			(* Case 157 - Attesa distacco lastra *)					
			157:
				IF Programma_Z[Z_PosDistaccoLastraInLentaLastra].Stato = INTERROTTO	THEN
					Ciclo^.Passo := 157;																
				ELSE
					TFTimerSet(ADR(TimerAttesaCadutaLastra),HMI_TempoAttesaPartenzaDopoPrelievo, Programma_Z[Z_PosDistaccoLastraInLentaLastra].Stato <> TERMINATO);		
					IF Programma_Z[Z_PosDistaccoLastraInLentaLastra].Stato = TERMINATO AND TFTimerDone(ADR(TimerAttesaCadutaLastra)) THEN
						TFParametersArrayClear(ADR(ParametersArray));
						TFCommandSend(CmdCheckPresence,ParametersArray,Modules^.Pinza.Cmd);
						Ciclo^.Passo := 158;	
					END_IF
				END_IF	
					
			(* Case 158 -  Attesa completamento del comando *)
			158: 
				IF Programma_Z[Z_PosDistaccoLastraInLentaLastra].Stato = INTERROTTO	THEN
					Ciclo^.Passo := 158;																
				ELSE
					//TFTimerSet(ADR(TimerAttesaCadutaLastra),HMI_TempoAttesaPartenzaDopoPrelievo, (Programma_Z[Z_PosDistaccoLastraInLentaLastra].Stato <> TERMINATO));
					IF Programma_Z[Z_PosDistaccoLastraInLentaLastra].Stato = TERMINATO AND 
						TFTimerDone(ADR(TimerAttesaCadutaLastra)) AND
						TFStateCodeGet(Modules^.Pinza.State) = StateCHECKPRESENCE_END THEN
						IF Modules^.Pinza.StatoPinza.ElementoPrelevato THEN
							Ciclo^.Passo := 1000;	//CICLO TERMINATO
							Modules^.Ax_J.IN_Stop := TRUE; //Fermo Comando di tasteggio
							STEPDone := FALSE;
						ELSIF NOT Modules^.Pinza.StatoPinza.ElementoPrelevato THEN
							//IF NumeroTentativiPresaAttuali >= NumeroTentativiPresa THEN
								Errore := ErrMalfunzionamentoSensoriPresenzaPinza;
								//IF StepInto THEN
								//	Ciclo^.Passo 		:= 1000;//CICLO TERMINATO
								//	STEPDone 			:= FALSE;
								//END_IF
							//ELSE
								//Ciclo^.Passo := 150;//torno a fare prelievo
							//	NumeroTentativiPresaAttuali := NumeroTentativiPresaAttuali+1;
							//END_IF
						END_IF	
					END_IF
				END_IF	

			(* Case 1000 *)
			1000:
				STEPDone := TRUE;
				Ciclo^.Stato := TERMINATO;
				Ciclo^.Passo := 1000;
				
			(* Case 9999 - Ciclo NON annullato o NON terminato*)
			9999:
				Ciclo^.Stato := INTERROTTO;
				Ciclo^.Passo := 9999;
	ELSE						
		;	
	END_CASE;
ELSE								//Se il ciclo deve essere interrotto, setto il suo nuovo stato
	Ciclo^.Stato := INTERROTTO;
END_IF
END_ACTION

ACTION Verticale:
TFTimerCall(ADR(TimerAttesaCadutaLastra),TimeBase);
TFTimerCall(ADR(ReControlPiezaCogida),TimeBase); 
TFTimerCall(ADR(ReMovEjeX),TimeBase); 
(* Set della variabile che mi permette di fare lo STEP nel ciclo *)
StepInto := (Abilita_Ciclo_Step AND Command_Step) OR NOT Abilita_Ciclo_Step;

(* Reset Anticipo Dinamico se non ho l'abilitazione *)
IF NOT AbilitazioneAnticipoDinamicoMovimenti OR NOT HMI_DisabilitaAnticipiGLOBALE THEN
	QuotaAnticipoDinamicaX_Raggiunta := FALSE;
	QuotaAnticipoDinamicaY_Raggiunta := FALSE;
	QuotaAnticipoDinamicaZ_Raggiunta := FALSE;
END_IF
//
//
AttivazioneVuotoDistanza := TRUE;

IF Ciclo^.Passo = 116 THEN
Temp_INT[9] := 	Temp_INT[9] + 1;
TFTimerSet(ADR(ReControlPiezaCogida),10000, FALSE );	
ELSE
TFTimerSet(ADR(ReControlPiezaCogida),10000, TRUE );	
END_IF

IF Ciclo^.Passo = 27 THEN

TFTimerSet(ADR(ReMovEjeX),1000, FALSE );	
ELSE
TFTimerSet(ADR(ReMovEjeX),1000, 
TFAsseInFinestra(Posizione_Attuale := Modules^.AX_Y.Ax^.AxRef^.NcToPlc.ActPos ,
 Posizione_Finale := Programma_Y[Y_PosFuoriIngombroVuotoLastra].Quota_Destinazione ,FinestraDiControllo := 30.0 ) );	
END_IF

EjeYPosFueraIngombro := TFAsseInFinestra(Posizione_Attuale := Modules^.AX_Y.Ax^.AxRef^.NcToPlc.ActPos ,
 Posizione_Finale := Programma_Y[Y_PosFuoriIngombroVuotoLastra].Quota_Destinazione ,FinestraDiControllo := 30.0 );

EjeYPos0Ingombro :=  TFAsseInFinestra(Posizione_Attuale := Modules^.AX_Y.Ax^.AxRef^.NcToPlc.ActPos ,
 Posizione_Finale := Programma_Y[Y_PosPasillo0grados].Quota_Destinazione ,FinestraDiControllo := 30.0 ) ;
 
EjeYPos180Ingombro := TFAsseInFinestra(Posizione_Attuale := Modules^.AX_Y.Ax^.AxRef^.NcToPlc.ActPos ,
 Posizione_Finale := Programma_Y[Y_PosPasillo180grados].Quota_Destinazione ,FinestraDiControllo := 30.0 ) ;





Temp_Bool[58]:= TFAsseInFinestra(Posizione_Attuale := Modules^.AX_Y.Ax^.AxRef^.NcToPlc.ActPos ,
 Posizione_Finale := Programma_Y[Y_PosFuoriIngombroVuotoLastra].Quota_Destinazione ,FinestraDiControllo := 30.0 ) OR

(( TFAsseInFinestra(Posizione_Attuale := Modules^.AX_Y.Ax^.AxRef^.NcToPlc.ActPos ,
 Posizione_Finale := Programma_Y[Y_PosPasillo0grados].Quota_Destinazione ,FinestraDiControllo := 30.0 ) OR

TFAsseInFinestra(Posizione_Attuale := Modules^.AX_Y.Ax^.AxRef^.NcToPlc.ActPos ,
 Posizione_Finale := Programma_Y[Y_PosPasillo180grados].Quota_Destinazione ,FinestraDiControllo := 30.0 )) (*AND RobotWorkAreaCavallete (*AND MultiplesCavalletesReceta *) *))  ;

 
 
 
Temp_Bool[25] := TFTimerDone(ADR(ReControlPiezaCogida));

//Valuto l'angolo di J per stabilire se è "inclinata"

PinzaVerticale 	:= Modules^.AX_J.Ax^.Status.ActPosition > 95 OR Modules^.AX_J.Ax^.Status.ActPosition < 85;
PinzaInPresa	:= Modules^.Pinza.StatoPinza.LatoDxPiastrellaInPresa AND Modules^.Pinza.StatoPinza.LatoSxPiastrellaInPresa;


IF NOT InterrompiCiclo THEN
	IF Ciclo^.Stato = TERMINATO OR Ciclo^.Stato = ANNULLATO THEN
		Ciclo^.Passo 	:= 0;
		Errore 			:= 0;
	ELSIF Ciclo^.Stato = INTERROTTO THEN
		Ciclo^.Passo 	:= 9999;
	END_IF
	CASE Ciclo^.Passo OF

			(* Case 0 *)
			0:  Ciclo^.Stato 		:= IN_ESECUZIONE;
				ReqStartAspirazione := FALSE;
				STEPDone 			:= FALSE;
				PosicionJSalida    := 0 ;
				
				IF Modules^.Pinza.CmdNext.Code = '' AND NOT PinzaInPresa THEN
					TFParametersArrayClear(ADR(ParametersArray));
					IF InWaitPosition THEN
						Modules^.Pinza.IN.RichiestaRicalibrazioneOvemEsterna := TRUE; //Ricalibrazione automatica OVEM
					END_IF
					TFCommandSend(CmdUNLOAD,ParametersArray,Modules^.Pinza.Cmd);
					Ciclo^.Passo := 11;
				ELSIF PinzaInPresa THEN
					Errore := ErrPRESENZA_MATERIALE_SUPINZA_CICLO_PRELPACCO;
				END_IF
				(* Start tempo ciclo *)
				
			(* Case 11 - Attesa comando temrinato pinza *)
			11:			
				IF TFStateCodeGet(Modules^.Pinza.State) = StateUNLOAD_END THEN
					Ciclo^.Passo := 12;	
				ELSIF TFStateCodeGet(Modules^.Pinza.State) = StateError THEN
					Ciclo^.Passo := 11;																
				END_IF
				
			(* Case 12 - Blocca Rotazione e Basculante *)
			12:
				IF TFStateCodeGet(Modules^.Pinza.State) = StateError THEN
					Ciclo^.Passo := 12;																
				ELSE
					//TFParametersArrayClear(ADR(ParametersArray));
					//TFCommandSend(CmdBloccaPinza,ParametersArray,Modules^.Pinza.Cmd);
					Ciclo^.Passo := 13;
				END_IF				

			(* Case 13 - Blocca Rotazione e Basculante *)
			13:
				IF TFStateCodeGet(Modules^.Pinza.State) = StateError THEN
					Ciclo^.Passo := 13;																
				ELSE
					//IF TFStateCodeGet(Modules^.Pinza.State) = StateBloccaPinza_END THEN//Pinza bloccata
						Ciclo^.Passo := 20;
					//END_IF	
				END_IF	
	
			(* Case 20 - TRASLAZIONE A QUOTA DI FUORI INGOMBRO *)	
			20:	
				//IF TFStateCodeGet(Modules^.Pinza.State) = StateUNLOAD_END THEN
					IF StepInto THEN
						Programma_Z[Z_PosFuoriIngombroVuotoLastra].Stato 			:= DA_ESEGUIRE;
						Programma_Z[Z_PosFuoriIngombroVuotoLastra].InterpolaAsse 	:= NO_INTERPOLAZIONE_ASSE;
						ProgrammaToModule_Z 										:= Programma_Z[Z_PosFuoriIngombroVuotoLastra];
						Ciclo^.Passo := 21;
						STEPDone := FALSE;
						
					(*	Programma_Z[Z_PosFuoriIngombroCaricoLastra].Stato 			:= DA_ESEGUIRE;
						Programma_Z[Z_PosFuoriIngombroCaricoLastra].InterpolaAsse 	:= NO_INTERPOLAZIONE_ASSE;
						ProgrammaToModule_Z 										:= Programma_Z[Z_PosFuoriIngombroCaricoLastra];
						Ciclo^.Passo := 21;
						STEPDone := FALSE; *)
					END_IF
				//END_IF
				
			(* Case 21 - Attesa completamento del comando MOVETOPOS o del raggiungimento quota di Pre-Movimento se abilitata la funzione*)
			21: 
					
				//IF Programma_Z[Z_PosFuoriIngombroCaricoLastra].Stato = INTERROTTO THEN
				IF Programma_Z[Z_PosFuoriIngombroVuotoLastra].Stato = INTERROTTO THEN
					Ciclo^.Passo := 21;		
				//ELSIF Programma_Z[Z_PosFuoriIngombroCaricoLastra].Stato = TERMINATO OR
				ELSIF Programma_Z[Z_PosFuoriIngombroVuotoLastra].Stato = TERMINATO OR
					Asse_Z_InFinestraDiPassMode THEN
					IF PinzaVerticale THEN//Se la pinza è già verticale in finestra di prelievo

						IF Modules^.AX_Y.Ax^.AxRef^.NcToPlc.ActPos <= Programma_Y[Y_PosFuoriIngombroVuotoLastra].Quota_Destinazione AND NOT RobotWorkAreaCavallete THEN
							Programma_Y[Y_PosFuoriIngombroVuotoLastra].Stato 				:= DA_ESEGUIRE;
							//Programma_Y[Y_PosFuoriIngombroVuotoLastra].InterpolaAsse 		:= INTERPOLAZIONE_ASSE;
							Programma_Y[Y_PosFuoriIngombroVuotoLastra].InterpolaAsse 		:= No_INTERPOLAZIONE_ASSE;
							ProgrammaToModule_Y 									:= Programma_Y[Y_PosFuoriIngombroVuotoLastra];
							
							Programma_J[J_PosFuoriIngombroPosAttuale].Stato 		:= DA_ESEGUIRE;
							//Programma_J[J_PosFuoriIngombroPosAttuale].InterpolaAsse := INTERPOLAZIONE_ASSE;
							Programma_J[J_PosFuoriIngombroPosAttuale].InterpolaAsse := No_INTERPOLAZIONE_ASSE;
							ProgrammaToModule_J 									:= Programma_J[J_PosFuoriIngombroPosAttuale];
	
							StartInterpolazioneAssi^ 								:= TRUE;
							Ciclo^.Passo := 22; 
							STEPDone := TRUE;	
						ELSE
							Ciclo^.Passo := 23; 
							STEPDone := TRUE;	
						END_IF						
					ELSIF NOT PinzaVerticale THEN
						Ciclo^.Passo := 25; 
						STEPDone := TRUE;							
					ELSE
						Ciclo^.Passo := 21;		
						Errore := 1;
					END_IF
				END_IF
			
			(* Case 21 - Rotazione Asse K *)	
			22: IF Programma_Z[Z_PosFuoriIngombroVuotoLastra].Stato = INTERROTTO OR
					Programma_Y[Y_PosFuoriIngombroVuotoLastra].Stato = INTERROTTO OR
					Programma_J[J_PosFuoriIngombroPosAttuale].Stato = INTERROTTO THEN
					 Ciclo^.Passo := 22;
				ELSIF Programma_Z[Z_PosFuoriIngombroVuotoLastra].Stato = TERMINATO AND //OR Asse_Z_InFinestraDiPassMode) AND 
					Programma_Y[Y_PosFuoriIngombroVuotoLastra].Stato = TERMINATO AND//OR Asse_Y_InFinestraDiPassMode) AND
					Programma_J[J_PosFuoriIngombroPosAttuale].Stato = TERMINATO THEN//OR Asse_J_InFinestraDiPassMode) THEN
						IF StepInto THEN
							Ciclo^.Passo := 23;
							STEPDone := FALSE;
						END_IF									
				END_IF

			(* Case 23 - Attesa completamento comandi *)	
			23: 	
				STEPDone := TRUE;
				Ciclo^.Passo := 24;
	
			(* Case 24 - free *)	
			24:	
				STEPDone := FALSE;
				Ciclo^.Passo := 25;
			
			(* Case 25 - Vado a quota di CORRIDOIO PER ROTAZIONE con Y *)
			25:	IF Programma_Z[Z_PosFuoriIngombroVuotoLastra].Stato = INTERROTTO THEN
					Ciclo^.Passo := 25;										
				ELSE
					
					IF StepInto THEN
							//IF 	Programma_Z[Y_PosFuoriIngombroVuotoLastra].Stato = TERMINATO THEN
							IF 	Programma_Z[Z_PosFuoriIngombroVuotoLastra].Stato = TERMINATO  THEN
								PruLineaContactos := (PosRobot = NuPosGuiroPiking  AND PikingConCavallete) 
												OR (( NOT MultiplesCavalletesReceta 
												OR PosicionJDestino = PosicionJOrigen) AND NOT PikingConCavallete) ;
							
								
										
								(*
									Programma_X[X_PosStartLentaPrelievoLastra].Stato 			:= DA_ESEGUIRE;
									//Programma_X[X_PosStartLentaPrelievoLastra].InterpolaAsse 	:= INTERPOLAZIONE_ASSE;
									Programma_X[X_PosStartLentaPrelievoLastra].InterpolaAsse 	:= No_INTERPOLAZIONE_ASSE;
									ProgrammaToModule_X 										:= Programma_X[X_PosStartLentaPrelievoLastra];
								*)
								
								
								IF (AngulosDiferentes OR PosicionJDestino <> PosicionJActual)  AND (RobotWorkAreaCavallete OR MultiplesCavalletesReceta) THEN 
									Temp_UINT [1] := Temp_UINT [1]+1;
									IF PosicionJActual = 0 THEN
										(*
										//********************************************************************
										Programma_Y[Y_PosFuoriIngombroVuotoLastra].Stato 	:= NON_ESEGUITO;
										Programma_Y[Y_PosPasillo180grados].Stato 			:= NON_ESEGUITO;
										Programma_Y[Y_PosgiroPieza].Stato 					:= NON_ESEGUITO ;
										//*********************************************************************
										*)
										Programma_Y[Y_PosPasillo0grados].Stato 			:= DA_ESEGUIRE;
										Programma_Y[Y_PosPasillo0grados].InterpolaAsse 	:= INTERPOLAZIONE_ASSE;
										ProgrammaToModule_Y 							:= Programma_Y[Y_PosPasillo0grados];
										
										Programma_J[Pos0TrasporteCavallete].Stato 						:= DA_ESEGUIRE;
										Programma_J[Pos0TrasporteCavallete].InterpolaAsse 				:= No_INTERPOLAZIONE_ASSE;
										ProgrammaToModule_J 											:= Programma_J[Pos0TrasporteCavallete];	
										IF Temp_Bool[50] THEN
											StartInterpolazioneAssi^ := TRUE;
											Ciclo^.Passo := 27;
										END_IF
										
									END_IF
									IF PosicionJActual = 180 THEN
										Programma_Y[Y_PosPasillo180grados].Stato 			:= DA_ESEGUIRE;
										Programma_Y[Y_PosPasillo180grados].InterpolaAsse 	:= INTERPOLAZIONE_ASSE;
										ProgrammaToModule_Y 								:= Programma_Y[Y_PosPasillo180grados];
										
										Programma_J[Pos180TrasporteCavallete].Stato 						:= DA_ESEGUIRE;
										Programma_J[Pos180TrasporteCavallete].InterpolaAsse 				:= No_INTERPOLAZIONE_ASSE;
										ProgrammaToModule_J 											:= Programma_J[Pos180TrasporteCavallete];
										IF Temp_Bool[50] THEN
											StartInterpolazioneAssi^ := TRUE;
											Ciclo^.Passo := 27;
										END_IF
									END_IF
									
									IF PosicionJActual = 90 AND PosicionJOrigen = 0 THEN
										Programma_Y[Y_PosPasillo0grados].Stato 			:= DA_ESEGUIRE;
										Programma_Y[Y_PosPasillo0grados].InterpolaAsse 	:= INTERPOLAZIONE_ASSE;
										ProgrammaToModule_Y 								:= Programma_Y[Y_PosPasillo0grados];
										
										Programma_J[Pos0TrasporteCavallete].Stato 						:= DA_ESEGUIRE;
										Programma_J[Pos0TrasporteCavallete].InterpolaAsse 				:= No_INTERPOLAZIONE_ASSE;
										ProgrammaToModule_J 											:= Programma_J[Pos0TrasporteCavallete];
										IF Temp_Bool[50] THEN
											StartInterpolazioneAssi^ := TRUE;
											Ciclo^.Passo := 27;
										END_IF
									END_IF
									IF PosicionJActual = 90 AND PosicionJOrigen = 180 THEN
										Programma_Y[Y_PosPasillo180grados].Stato 			:= DA_ESEGUIRE;
										Programma_Y[Y_PosPasillo180grados].InterpolaAsse 	:= INTERPOLAZIONE_ASSE;
										ProgrammaToModule_Y 								:= Programma_Y[Y_PosPasillo180grados];
										
										Programma_J[Pos180TrasporteCavallete].Stato 						:= DA_ESEGUIRE;
										Programma_J[Pos180TrasporteCavallete].InterpolaAsse 				:= No_INTERPOLAZIONE_ASSE;
										ProgrammaToModule_J 											:= Programma_J[Pos180TrasporteCavallete];
										IF Temp_Bool[50] THEN
											StartInterpolazioneAssi^ := TRUE;
											Ciclo^.Passo := 27;
										END_IF
									END_IF
									//PosicionJSalida := PosicionJActual ;
								ELSIF NOT AngulosDiferentes AND RobotWorkAreaCavallete AND PosicionJDestino = PosicionJActual  THEN
										Temp_UINT [2] := Temp_UINT [2]+1;
										Programma_Y[Y_PosFuoriIngombroVuotoLastra].Stato 				:= DA_ESEGUIRE;
										Programma_Y[Y_PosFuoriIngombroVuotoLastra].InterpolaAsse 		:= No_INTERPOLAZIONE_ASSE;
										//Programma_Y[Y_PosFuoriIngombroVuotoLastra].InterpolaAsse 		:= INTERPOLAZIONE_ASSE;
										ProgrammaToModule_Y 										:= Programma_Y[Y_PosFuoriIngombroVuotoLastra];
										
										Programma_J[J_PosFuoriIngombro].Stato 						:= DA_ESEGUIRE;
										//Programma_J[J_PosFuoriIngombro].InterpolaAsse 				:= INTERPOLAZIONE_ASSE;
										Programma_J[J_PosFuoriIngombro].InterpolaAsse 				:= No_INTERPOLAZIONE_ASSE;
										ProgrammaToModule_J 										:= Programma_J[J_PosFuoriIngombro];
										IF Temp_Bool[50] THEN
											StartInterpolazioneAssi^ := TRUE;
											Ciclo^.Passo := 27;
										END_IF
										
								ELSIF  (PosRobot = NuPosGuiroPiking  AND PikingConCavallete) OR (( NOT MultiplesCavalletesReceta OR PosicionJDestino = PosicionJOrigen) AND NOT PikingConCavallete)   THEN
										Temp_UINT [3] := Temp_UINT [3]+1;
								
										Programma_Y[Y_PosFuoriIngombroVuotoLastra].Stato 				:= DA_ESEGUIRE;
										Programma_Y[Y_PosFuoriIngombroVuotoLastra].InterpolaAsse 		:= No_INTERPOLAZIONE_ASSE;
										//Programma_Y[Y_PosFuoriIngombroVuotoLastra].InterpolaAsse 		:= INTERPOLAZIONE_ASSE;
										ProgrammaToModule_Y 										:= Programma_Y[Y_PosFuoriIngombroVuotoLastra];
										
										Programma_J[J_PosFuoriIngombro].Stato 						:= DA_ESEGUIRE;
										//Programma_J[J_PosFuoriIngombro].InterpolaAsse 				:= INTERPOLAZIONE_ASSE;
										Programma_J[J_PosFuoriIngombro].InterpolaAsse 				:= No_INTERPOLAZIONE_ASSE;
										ProgrammaToModule_J 										:= Programma_J[J_PosFuoriIngombro];		
										IF Temp_Bool[50] THEN
											StartInterpolazioneAssi^ := TRUE;
											Ciclo^.Passo := 27;
										END_IF
								ELSIF (AngulosDiferentes OR PosicionJDestino <> PosicionJActual)  AND WorkAreaState[PosRobot].Supporto.Tipologia <> CAVALLETTO AND  PikingConCavallete AND  NuPosGuiroPiking <> PosRobot  THEN
									Temp_UINT [4] := Temp_UINT [4]+1;	
									IF PosicionJOrigen = 0 THEN
											
										(*
										//********************************************************************
										Programma_Y[Y_PosFuoriIngombroVuotoLastra].Stato 	:= NON_ESEGUITO;
										Programma_Y[Y_PosPasillo180grados].Stato 			:= NON_ESEGUITO;
										Programma_Y[Y_PosgiroPieza].Stato 					:= NON_ESEGUITO ;
										//*********************************************************************
										*)
										Programma_Y[Y_PosPasillo0grados].Stato 			:= DA_ESEGUIRE;
										Programma_Y[Y_PosPasillo0grados].InterpolaAsse 	:= INTERPOLAZIONE_ASSE;
										ProgrammaToModule_Y 							:= Programma_Y[Y_PosPasillo0grados];
										
										Programma_J[Pos0TrasporteCavallete].Stato 						:= DA_ESEGUIRE;
										Programma_J[Pos0TrasporteCavallete].InterpolaAsse 				:= No_INTERPOLAZIONE_ASSE;
										ProgrammaToModule_J 											:= Programma_J[Pos0TrasporteCavallete];	
										IF Temp_Bool[50] THEN
											StartInterpolazioneAssi^ := TRUE;
											Ciclo^.Passo := 27;
										END_IF
										
									END_IF
									IF PosicionJOrigen = 180 THEN
										Programma_Y[Y_PosPasillo180grados].Stato 			:= DA_ESEGUIRE;
										Programma_Y[Y_PosPasillo180grados].InterpolaAsse 	:= INTERPOLAZIONE_ASSE;
										ProgrammaToModule_Y 								:= Programma_Y[Y_PosPasillo180grados];
										
										Programma_J[Pos180TrasporteCavallete].Stato 						:= DA_ESEGUIRE;
										Programma_J[Pos180TrasporteCavallete].InterpolaAsse 				:= No_INTERPOLAZIONE_ASSE;
										ProgrammaToModule_J 											:= Programma_J[Pos180TrasporteCavallete];
										IF Temp_Bool[50] THEN
											StartInterpolazioneAssi^ := TRUE;
											Ciclo^.Passo := 27;
										END_IF
									END_IF
								END_IF
						END_IF
					END_IF
				END_IF
			27:	 
				Temp_Bool[84] := 
							PosicionJOrigen = PosicionJActual OR NOT MultiplesCavalletesReceta	 ; 
				Temp_Bool[99]:= Programma_Y[Y_PosFuoriIngombroVuotoLastra].Stato = TERMINATO AND 
						Programma_Z[Z_PosFuoriIngombroVuotoLastra].Stato = TERMINATO AND 
						(Programma_J[J_PosFuoriIngombro].Stato = TERMINATO OR     
						(Programma_J[Pos0TrasporteCavallete].Stato = TERMINATO AND PosicionJOrigen = 0 ) OR
						(Programma_J[Pos180TrasporteCavallete].Stato = TERMINATO AND PosicionJOrigen = 180) OR 
							(PosicionJOrigen = PosicionJActual OR NOT MultiplesCavalletesReceta) ); 
					
		IF  ((Programma_Y[Y_PosFuoriIngombroVuotoLastra].Stato = INTERROTTO AND ProgramaEjes.EjeY = 106) OR 
			(Programma_Y[Y_PosPasillo0grados].Stato = INTERROTTO AND ProgramaEjes.EjeY = 128) OR 
			(Programma_Y[Y_PosPasillo180grados].Stato = INTERROTTO AND ProgramaEjes.EjeY = 129) OR 
			(Programma_J[J_PosFuoriIngombro].Stato = INTERROTTO AND ProgramaEjes.EjeJ = 6    ) OR 
			(Programma_J[Pos0TrasporteCavallete].Stato = INTERROTTO AND ProgramaEjes.EjeJ = 0    )OR 
			(Programma_J[Pos180TrasporteCavallete].Stato = INTERROTTO AND ProgramaEjes.EjeJ = 180  )OR
			Programma_Z[Z_PosFuoriIngombroVuotoLastra].Stato = INTERROTTO  )	
			 (* AND PosicionJDestino = PosicionJActual*) THEN  
			Ciclo^.Passo := 27;
					
			
		ELSE	
				//IF PosicionJDestino <> PosicionJActual AND  PosRobot <> NuPosGuiroPiking  THEN
				IF PosicionJOrigen <> PosicionJActual AND  PosRobot <> NuPosGuiroPiking AND NuPosGuiroPiking <> 0  THEN
					IF (EjeYPos0Ingombro OR EjeYPos180Ingombro) AND Temp_Bool[57] THEN 
					Programma_X[X_PosGiroPiezaTraCavallete].Stato 			:= DA_ESEGUIRE;
					Programma_X[X_PosGiroPiezaTraCavallete].InterpolaAsse 	:= No_INTERPOLAZIONE_ASSE;
					ProgrammaToModule_X 									:= Programma_X[X_PosGiroPiezaTraCavallete];
					Ciclo^.Passo := 31;
					END_IF
				ELSE 
					IF EjeYPosFueraIngombro OR (ProgramaEjes.EjeY = 128 AND EjeYPos0Ingombro) OR  (ProgramaEjes.EjeY = 129 AND EjeYPos180Ingombro)
									AND Temp_Bool[51] THEN
						Programma_X[X_PosStartLentaPrelievoLastra].Stato 			:= DA_ESEGUIRE;
						Programma_X[X_PosStartLentaPrelievoLastra].InterpolaAsse 	:= No_INTERPOLAZIONE_ASSE;
						ProgrammaToModule_X 										:= Programma_X[X_PosStartLentaPrelievoLastra];
						Ciclo^.Passo := 28;
					END_IF
								
				END_IF
		END_IF	
			
			(*
			
			27:	 
				Temp_Bool[84] := 
							PosicionJOrigen = PosicionJActual OR NOT MultiplesCavalletesReceta	 ; 
				Temp_Bool[99]:= Programma_Y[Y_PosFuoriIngombroVuotoLastra].Stato = TERMINATO AND 
						Programma_Z[Z_PosFuoriIngombroVuotoLastra].Stato = TERMINATO AND 
						(Programma_J[J_PosFuoriIngombro].Stato = TERMINATO OR     
						(Programma_J[Pos0TrasporteCavallete].Stato = TERMINATO AND PosicionJOrigen = 0 ) OR
						(Programma_J[Pos180TrasporteCavallete].Stato = TERMINATO AND PosicionJOrigen = 180) OR 
							(PosicionJOrigen = PosicionJActual OR NOT MultiplesCavalletesReceta) ); 
					
				IF  Programma_Y[Y_PosFuoriIngombroVuotoLastra].Stato = INTERROTTO OR 
					Programma_Z[Z_PosFuoriIngombroVuotoLastra].Stato = INTERROTTO OR 
					Programma_J[J_PosFuoriIngombro].Stato = INTERROTTO OR  
					((Programma_J[Pos0TrasporteCavallete].Stato = INTERROTTO  OR
					Programma_J[Pos180TrasporteCavallete].Stato = INTERROTTO) AND NOT  Programma_J[J_PosFuoriIngombro].Stato = TERMINATO) THEN
					Ciclo^.Passo := 27;
					
								
				ELSIF 
						(*
						Programma_Y[Y_PosFuoriIngombroVuotoLastra].Stato = TERMINATO AND 
						Programma_Z[Z_PosFuoriIngombroVuotoLastra].Stato = TERMINATO AND 
						(Programma_J[J_PosFuoriIngombro].Stato = TERMINATO AND  
						(Programma_J[Pos0TrasporteCavallete].Stato = TERMINATO AND PosicionJOrigen = 0 OR
						Programma_J[Pos180TrasporteCavallete].Stato = TERMINATO AND PosicionJOrigen = 180)) OR 
							PosicionJOrigen = PosicionJActual OR NOT MultiplesCavalletesReceta  THEN 
						*)
						
						
						
						
						
						Programma_Y[Y_PosFuoriIngombroVuotoLastra].Stato = TERMINATO AND 
						Programma_Z[Z_PosFuoriIngombroVuotoLastra].Stato = TERMINATO AND 
						(Programma_J[J_PosFuoriIngombro].Stato = TERMINATO OR     
						(Programma_J[Pos0TrasporteCavallete].Stato = TERMINATO AND PosicionJOrigen = 0 ) OR
						(Programma_J[Pos180TrasporteCavallete].Stato = TERMINATO AND PosicionJOrigen = 180) OR 
							(PosicionJOrigen = PosicionJActual OR NOT MultiplesCavalletesReceta) ) THEN 
							IF PosicionJDestino <> PosicionJActual  THEN
								IF Temp_Bool[58] AND Temp_Bool[57] THEN 
								Programma_X[X_PosStartLentaPrelievoLastra].Stato 			:= DA_ESEGUIRE;
								Programma_X[X_PosStartLentaPrelievoLastra].InterpolaAsse 	:= No_INTERPOLAZIONE_ASSE;
								ProgrammaToModule_X 										:= Programma_X[X_PosStartLentaPrelievoLastra];
								Ciclo^.Passo := 28;
								END_IF
							ELSE 
								IF Temp_Bool[58] AND Temp_Bool[51] THEN
									Programma_X[X_PosStartLentaPrelievoLastra].Stato 			:= DA_ESEGUIRE;
									Programma_X[X_PosStartLentaPrelievoLastra].InterpolaAsse 	:= No_INTERPOLAZIONE_ASSE;
									ProgrammaToModule_X 										:= Programma_X[X_PosStartLentaPrelievoLastra];
									Ciclo^.Passo := 28;
								END_IF
								
							END_IF
                                
					
				
		
				END_IF
			
			*)	
					
			(* Case 28 -  *)		

			28: (* Case 28 - Movimiento Pos Guiro *)
			
			
					
				IF Programma_X[X_PosStartLentaPrelievoLastra].Stato = INTERROTTO OR
					(Programma_Y[Y_PosFuoriIngombroVuotoLastra].Stato = INTERROTTO AND ProgramaEjes.EjeY = 106 ) OR 
					(Programma_Y[Y_PosPasillo0grados].Stato = INTERROTTO AND ProgramaEjes.EjeY = 128 ) OR 
					(Programma_Y[Y_PosPasillo180grados].Stato = INTERROTTO AND ProgramaEjes.EjeY = 129 ) OR 
					Programma_Z[Z_PosFuoriIngombroVuotoLastra].Stato = INTERROTTO OR 
					(Programma_J[Pos0TrasporteCavallete].Stato = INTERROTTO AND PosicionJSalida = 0 )OR
					(Programma_J[Pos180TrasporteCavallete].Stato = INTERROTTO AND PosicionJSalida = 180)  (*AND PosicionJSalida <> PosicionJDestino AND PosicionJDestino <> 90 *)THEN 
					Ciclo^.Passo := 28;
				ELSE	
					
					IF Programma_X[X_PosStartLentaPrelievoLastra].Stato = TERMINATO AND
						((Programma_Y[Y_PosFuoriIngombroVuotoLastra].Stato = TERMINATO AND ProgramaEjes.EjeY = 106 ) OR 
						(Programma_Y[Y_PosPasillo0grados].Stato = TERMINATO AND ProgramaEjes.EjeY = 128 ) OR 
						(Programma_Y[Y_PosPasillo180grados].Stato = TERMINATO AND ProgramaEjes.EjeY = 129 ) )
																								 AND 
						Programma_Z[Z_PosFuoriIngombroVuotoLastra].Stato = TERMINATO AND
						(Programma_J[Pos0TrasporteCavallete].Stato = TERMINATO AND PosicionJActual = 0 OR
						Programma_J[Pos180TrasporteCavallete].Stato = TERMINATO AND PosicionJActual = 180 OR PosicionJOrigen = PosicionJActual  ) (* AND PosicionJSalida <> PosicionJDestino AND PosicionJDestino <> 90*)
						AND TFAsseInFinestra(Posizione_Attuale := Modules^.AX_X.Ax^.AxRef^.NcToPlc.ActPos ,
 							Posizione_Finale := Programma_X[X_PosStartLentaPrelievoLastra].Quota_Destinazione ,FinestraDiControllo := 30.0 )
						AND Temp_Bool[100]  THEN 
						 IF PosicionJOrigen <> PosicionJActual  THEN
							// Muevo El Eje y Cota De giro pieza
								Programma_Y[Y_PosgiroPieza].Stato 				:= DA_ESEGUIRE;
								Programma_Y[Y_PosgiroPieza].InterpolaAsse 		:= No_INTERPOLAZIONE_ASSE;
								ProgrammaToModule_Y 							:= Programma_Y[Y_PosgiroPieza];
								IF Temp_Bool[53] THEN
									Ciclo^.Passo := 29;
									STEPDone := TRUE;
								END_IF
									
							
						ELSE
								Ciclo^.Passo := 26;
								STEPDone := TRUE;
						END_IF

						
						
					END_IF
				END_IF	

			29: (* Case 28 - Movimiento Pos Guiro *)
				IF Programma_X[X_PosStartLentaPrelievoLastra].Stato = INTERROTTO OR
					Programma_Y[Y_PosgiroPieza].Stato = INTERROTTO OR 
					Programma_Z[Z_PosFuoriIngombroVuotoLastra].Stato = INTERROTTO OR 
					(Programma_J[Pos0TrasporteCavallete].Stato = INTERROTTO AND PosicionJSalida = 0 )OR
					(Programma_J[Pos180TrasporteCavallete].Stato = INTERROTTO AND PosicionJSalida = 180)  AND PosicionJSalida <> PosicionJDestino AND PosicionJDestino <> 90 THEN 
						Ciclo^.Passo := 29;
				ELSE	
					IF Programma_X[X_PosStartLentaPrelievoLastra].Stato = TERMINATO AND
						Programma_Y[Y_PosgiroPieza].Stato 				= TERMINATO AND
						Programma_Z[Z_PosFuoriIngombroVuotoLastra].Stato = TERMINATO AND
						
						((Programma_J[Pos0TrasporteCavallete].Stato = TERMINATO AND PosicionJSalida = 0 )OR
						(Programma_J[Pos180TrasporteCavallete].Stato = TERMINATO AND PosicionJSalida = 180) ) AND PosicionJSalida <> PosicionJDestino AND PosicionJDestino <> 90 THEN 
						// Muevo El Eje J Cota De DejarPieza
						Programma_J[J_PosFuoriIngombro].Stato 						:= DA_ESEGUIRE;
						Programma_J[J_PosFuoriIngombro].InterpolaAsse 				:= No_INTERPOLAZIONE_ASSE;
						ProgrammaToModule_J 										:= Programma_J[J_PosFuoriIngombro];
						IF Temp_Bool[54] THEN
							Ciclo^.Passo := 30;
							STEPDone := TRUE;
						END_IF
						
					END_IF
				END_IF	
			30: (* Case 28 - Movimiento Pos Guiro *)
				IF Programma_X[X_PosStartLentaPrelievoLastra].Stato = INTERROTTO OR
					Programma_Y[Y_PosgiroPieza].Stato = INTERROTTO OR 
					Programma_Z[Z_PosFuoriIngombroVuotoLastra].Stato = INTERROTTO OR 
					Programma_J[J_PosFuoriIngombro].Stato = INTERROTTO THEN 
					Ciclo^.Passo := 30;
				ELSE	
					IF Programma_X[X_PosStartLentaPrelievoLastra].Stato = TERMINATO OR
						Programma_Y[Y_PosgiroPieza].Stato 				= TERMINATO OR 
						Programma_Z[Z_PosFuoriIngombroVuotoLastra].Stato = TERMINATO OR 
						Programma_J[J_PosFuoriIngombro].Stato 			= TERMINATO  THEN 
						IF Temp_Bool[55] THEN
							Ciclo^.Passo := 26;
						STEPDone := TRUE;
						END_IF
						
					END_IF
				END_IF	
				
			
			31: (* Case 28 - Movimiento Pos Transporte A-Frame Picking *)
				IF Programma_X[X_PosGiroPiezaTraCavallete].Stato = INTERROTTO OR
					(Programma_Y[Y_PosPasillo0grados].Stato = INTERROTTO OR Programma_Y[Y_PosPasillo180grados].Stato = INTERROTTO) OR
					Programma_Z[Z_PosFuoriIngombroVuotoLastra].Stato = INTERROTTO OR 
					(Programma_J[Pos180TrasporteCavallete].Stato = INTERROTTO  OR Programma_J[Pos0TrasporteCavallete].Stato = INTERROTTO) THEN 
					Ciclo^.Passo := 31;
				ELSE	
					IF Programma_X[X_PosGiroPiezaTraCavallete].Stato = TERMINATO AND 
						((Programma_Y[Y_PosPasillo0grados].Stato 	= TERMINATO AND PosicionJActual = 0) OR
						(Programma_Y[Y_PosPasillo180grados].Stato 	= TERMINATO AND PosicionJActual = 180)) AND 
						Programma_Z[Z_PosFuoriIngombroVuotoLastra].Stato = TERMINATO AND
						((Programma_J[Pos0TrasporteCavallete].Stato 			= TERMINATO AND PosicionJOrigen = 0) OR
						(Programma_J[Pos180TrasporteCavallete].Stato 			= TERMINATO AND PosicionJOrigen = 180))	THEN 
						
						IF WorkAreaState[PosRobot].Supporto.Tipologia = BUNDLE AND PosicionJActual <> PosicionJDestino THEN
							
							Programma_Y[Y_PosgiroPieza].Stato 			:= DA_ESEGUIRE;
							Programma_Y[Y_PosgiroPieza].InterpolaAsse 	:= INTERPOLAZIONE_ASSE;
							ProgrammaToModule_Y 										:= Programma_Y[Y_PosgiroPieza];
							
							Programma_J[J_PosFuoriIngombro].Stato 						:= DA_ESEGUIRE;
							Programma_J[J_PosFuoriIngombro].InterpolaAsse 				:= No_INTERPOLAZIONE_ASSE;
							ProgrammaToModule_J 										:= Programma_J[J_PosFuoriIngombro];	
							IF Temp_Bool[55]  THEN
								Ciclo^.Passo := 32;
								STEPDone := TRUE;
							END_IF
						ELSE
							Programma_Y[Y_PosFuoriIngombroVuotoLastra].Stato 			:= DA_ESEGUIRE;
							Programma_Y[Y_PosFuoriIngombroVuotoLastra].InterpolaAsse 	:= INTERPOLAZIONE_ASSE;
							ProgrammaToModule_Y 							:= Programma_Y[Y_PosFuoriIngombroVuotoLastra];
											
							Programma_J[J_PosFuoriIngombro].Stato 						:= DA_ESEGUIRE;
							Programma_J[J_PosFuoriIngombro].InterpolaAsse 				:= No_INTERPOLAZIONE_ASSE;
							ProgrammaToModule_J 										:= Programma_J[J_PosFuoriIngombro];	
								
							IF Temp_Bool[55]  THEN
								Ciclo^.Passo := 27;
								STEPDone := TRUE;
							END_IF
						END_IF
						
						
						
					END_IF
				END_IF	

			32: (* Añadido Trabajo Bundel  *)

				IF Programma_X[X_PosGiroPiezaTraCavallete].Stato = TERMINATO AND 
						Programma_Y[Y_PosgiroPieza].Stato 	= TERMINATO AND  
							Programma_Z[Z_PosFuoriIngombroVuotoLastra].Stato = TERMINATO AND
								Programma_J[Pos0TrasporteCavallete].Stato 			= TERMINATO  THEN 
						
							Programma_Y[Y_PosFuoriIngombroVuotoLastra].Stato 			:= DA_ESEGUIRE;
							Programma_Y[Y_PosFuoriIngombroVuotoLastra].InterpolaAsse 	:= INTERPOLAZIONE_ASSE;
							ProgrammaToModule_Y 										:= Programma_Y[Y_PosFuoriIngombroVuotoLastra];
											
							
								
							IF Temp_Bool[55]  THEN
								Ciclo^.Passo := 27;
								STEPDone := TRUE;
							END_IF
						
						END_IF
	
				
			26:	
					

				IF Programma_X[X_PosStartLentaPrelievoLastra].Stato = INTERROTTO OR
					(Programma_Y[Y_PosFuoriIngombroVuotoLastra].Stato = INTERROTTO AND ProgramaEjes.EjeY = 106 ) OR 
					(Programma_Y[Y_PosPasillo0grados].Stato = INTERROTTO AND ProgramaEjes.EjeY = 128 ) OR 
					(Programma_Y[Y_PosPasillo180grados].Stato = INTERROTTO AND ProgramaEjes.EjeY = 129 ) OR 
					(Programma_Y[Y_PosgiroPieza].Stato = INTERROTTO AND ProgramaEjes.EjeY = 127 ) OR 
					Programma_Z[Z_PosFuoriIngombroVuotoLastra].Stato = INTERROTTO OR 
					(Programma_J[J_PosFuoriIngombro].Stato = INTERROTTO AND ProgramaEjes.EjeJ = 6) OR 
					(Programma_J[Pos0TrasporteCavallete].Stato = INTERROTTO AND ProgramaEjes.EjeJ = 0)OR  	
					(Programma_J[Pos180TrasporteCavallete].Stato = INTERROTTO AND ProgramaEjes.EjeJ = 180)  THEN
						Ciclo^.Passo := 26;
				ELSE	
					IF Programma_X[X_PosStartLentaPrelievoLastra].Stato = TERMINATO AND
						((Programma_Y[Y_PosFuoriIngombroVuotoLastra].Stato = TERMINATO AND ProgramaEjes.EjeY = 106 ) OR 
						(Programma_Y[Y_PosPasillo0grados].Stato = TERMINATO AND ProgramaEjes.EjeY = 128 ) OR 
						(Programma_Y[Y_PosPasillo180grados].Stato = TERMINATO AND ProgramaEjes.EjeY = 129 ) OR 
						(Programma_Y[Y_PosgiroPieza].Stato = TERMINATO AND ProgramaEjes.EjeY = 127 ))AND 
						Programma_Z[Z_PosFuoriIngombroVuotoLastra].Stato = TERMINATO AND 
						(Programma_J[J_PosFuoriIngombro].Stato = TERMINATO AND ProgramaEjes.EjeJ = 6 OR
								(( Programma_J[Pos0TrasporteCavallete].Stato = TERMINATO AND  ProgramaEjes.EjeJ = 0 OR 
										Programma_J[Pos180TrasporteCavallete].Stato = TERMINATO AND ProgramaEjes.EjeJ = 180)(*  AND 
												MultiplesCavalletesReceta AND  PikingConCavallete *))) THEN
							IF StepInto THEN
								Programma_Z[Z_PosStartLentaPrelievoLastra].Stato 			:= DA_ESEGUIRE;
								Programma_Z[Z_PosStartLentaPrelievoLastra].InterpolaAsse 	:= NO_INTERPOLAZIONE_ASSE;
								ProgrammaToModule_Z 										:= Programma_Z[Z_PosStartLentaPrelievoLastra];
								Ciclo^.Passo := 40;
								STEPDone := TRUE;
							END_IF
					END_IF
				END_IF
						
			(* Case 40 - *)
			40:
				Ciclo^.Passo := 41;
				STEPDone := FALSE;
				
			(* Case 41 - *)
			41:
				STEPDone 		:= TRUE;
				Ciclo^.Passo 	:= 42;

			(* Case 42 - Vado a quota di START LENTA CON GLI ASSI con Y,Z,J *)
			42:
				IF Programma_Z[Z_PosStartLentaPrelievoLastra].Stato = INTERROTTO THEN
					Ciclo^.Passo := 42;	
				ELSIF Programma_Z[Z_PosStartLentaPrelievoLastra].Stato = TERMINATO THEN
					TimerAttesaFiltroFtc(IN:=TRUE,PT:=T#1200MS);
					IF StepInto AND TimerAttesaFiltroFtc.Q THEN
						TFParametersArrayClear(ADR(ParametersArray));
						Programma_Y[Y_PosStartLentaPrelievoLastra].Stato 			:= DA_ESEGUIRE;
						Programma_Y[Y_PosStartLentaPrelievoLastra].InterpolaAsse 	:= INTERPOLAZIONE_ASSE;
						ProgrammaToModule_Y 										:= Programma_Y[Y_PosStartLentaPrelievoLastra];
				
						//Programma_Z[Z_PosStartLentaPrelievoLastra].Stato 			:= DA_ESEGUIRE;
						//Programma_Z[Z_PosStartLentaPrelievoLastra].InterpolaAsse 	:= INTERPOLAZIONE_ASSE;
						//ProgrammaToModule_Z 										:= Programma_Z[Z_PosStartLentaPrelievoLastra];
						//(* Aggiusto la quota del j con quella calcolata dalle ftc *)
						IF ABS(Programma_J[J_PosStartApproccioPrelLastra].Quota_Destinazione - Modules^.AX_J.QuotaAssePerPianoParallelo) <= 5 THEN
							IF HMI_OffsetGradiJPrelDaCanti > 0.5 THEN
								HMI_OffsetGradiJPrelDaCanti := 0;
							ELSIF HMI_OffsetGradiJPrelDaCanti < -0.5 THEN
								HMI_OffsetGradiJPrelDaCanti := -0.5;
							END_IF
							IF Programma_J[J_PosStartApproccioPrelLastra].Quota_Destinazione > 100 THEN
								//original
								//QuotaJPerAsseInPiano := Modules^.AX_J.QuotaAssePerPianoParallelo + HMI_OffsetGradiJPrelDaCanti + 0.2;
								QuotaJPerAsseInPiano := MIN (Programma_J[J_PosStartApproccioPrelLastra].Quota_Destinazione , Modules^.AX_J.QuotaAssePerPianoParallelo + HMI_OffsetGradiJPrelDaCanti + 0.2);
							ELSIF Programma_J[J_PosStartApproccioPrelLastra].Quota_Destinazione < 80 THEN
								QuotaJPerAsseInPiano :=MAX(Programma_J[J_PosStartApproccioPrelLastra].Quota_Destinazione, Modules^.AX_J.QuotaAssePerPianoParallelo + HMI_OffsetGradiJPrelDaCanti - 0.2);
							ELSE
								QuotaJPerAsseInPiano := Modules^.AX_J.QuotaAssePerPianoParallelo + HMI_OffsetGradiJPrelDaCanti;
							END_IF
							IF HMI_AbilitaPosJPrelConFTC THEN
								Programma_J[J_PosStartApproccioPrelLastra].Quota_Destinazione := QuotaJPerAsseInPiano;
							END_IF
						END_IF
	
						Programma_J[J_PosStartApproccioPrelLastra].Stato 			:= DA_ESEGUIRE;
						//Programma_J[J_PosStartApproccioPrelLastra].InterpolaAsse 	:= INTERPOLAZIONE_ASSE;
						Programma_J[J_PosStartApproccioPrelLastra].InterpolaAsse 	:= No_INTERPOLAZIONE_ASSE;
						ProgrammaToModule_J 										:= Programma_J[J_PosStartApproccioPrelLastra];
						
						StartInterpolazioneAssi^ 	:= TRUE; //Abilito l'interpolazione degli assi
											
						Ciclo^.Passo := 43;
						STEPDone := FALSE;
					END_IF
				END_IF
			
			(* Case 43 - *)
			43:
				TimerAttesaFiltroFtc(IN:=FALSE,PT:=T#1200MS);
				Ciclo^.Passo := 52;//50;
				
			(* Case 50 - ASSE Z -> TRASLAZIONE A QUOTA AMMESSA IN VELOCE DI PRELIEVO  *)
			50:
				IF Programma_Y[Y_PosStartLentaPrelievoLastra].Stato = INTERROTTO OR
					Programma_J[J_PosStartApproccioPrelLastra].Stato = INTERROTTO THEN
					Ciclo^.Passo := 50;
				ELSIF Programma_Y[Y_PosStartLentaPrelievoLastra].Stato = TERMINATO AND
					Programma_J[J_PosStartApproccioPrelLastra].Stato = TERMINATO THEN
						IF StepInto THEN
							Programma_Z[Z_PosStartLentaPrelievoLastra].Stato 			:= DA_ESEGUIRE;
							Programma_Z[Z_PosStartLentaPrelievoLastra].InterpolaAsse 	:= NO_INTERPOLAZIONE_ASSE;
							ProgrammaToModule_Z 										:= Programma_Z[Z_PosStartLentaPrelievoLastra];
							StartInterpolazioneAssi^									:= FALSE; //Abilito l'interpolazione degli assi
							Ciclo^.Passo := 52;
							STEPDone := FALSE;
						END_IF
				END_IF
			
			(* Case 52 -  *)
			52:
				IF Programma_Z[Z_PosStartLentaPrelievoLastra].Stato = INTERROTTO OR
					Programma_Y[Y_PosStartLentaPrelievoLastra].Stato = INTERROTTO OR
					Programma_J[J_PosStartApproccioPrelLastra].Stato = INTERROTTO THEN
						Ciclo^.Passo := 52;									
				ELSE
					IF Programma_Y[Y_PosStartLentaPrelievoLastra].Stato	= TERMINATO AND
						Programma_J[J_PosStartApproccioPrelLastra].Stato = TERMINATO AND
						Programma_Z[Z_PosStartLentaPrelievoLastra].Stato = TERMINATO THEN
							STEPDone := TRUE;
							IF StepInto THEN
								Programma_Z[Z_PosPrelievoInLentaLastra].Stato 			:= DA_ESEGUIRE;
								Programma_Z[Z_PosPrelievoInLentaLastra].InterpolaAsse 	:= NO_INTERPOLAZIONE_ASSE;
								ProgrammaToModule_Z 									:= Programma_Z[Z_PosPrelievoInLentaLastra];
								Ciclo^.Passo 	:= 53;
								STEPDone 		:= FALSE;
							END_IF
					END_IF	
				END_IF
			
			(* Case 53 -  *)						
			53:
				IF Programma_Z[Z_PosPrelievoInLentaLastra].Stato = INTERROTTO OR
					Programma_Y[Y_PosStartLentaPrelievoLastra].Stato = INTERROTTO OR
					Programma_J[J_PosStartApproccioPrelLastra].Stato = INTERROTTO THEN
						Ciclo^.Passo := 53;									
				ELSE
					IF Programma_Y[Y_PosStartLentaPrelievoLastra].Stato	= TERMINATO AND
						Programma_J[J_PosStartApproccioPrelLastra].Stato 	= TERMINATO AND
							(Programma_Z[Z_PosPrelievoInLentaLastra].Stato = TERMINATO )THEN
							Ciclo^.Passo := 90;
							STEPDone := TRUE;
					END_IF	
				END_IF
				
			(* Case 85 - *)
			85:
				Ciclo^.Passo := 86; 	
							
			(* Case 86 - *)
			86:
				Ciclo^.Passo := 90;
								

			(* Case 90 - PROGRAMMA[] ASSE Y -> TRASLAZIONE IN Y FINO ALLA QUOTA AMMESSA IN VELOCE E ATTIVAZIONE ASPIRAZIONE *)
			90:
				IF Programma_Z[Z_PosStartLentaPrelievoLastra].Stato = INTERROTTO OR
					Programma_Y[Y_PosStartLentaPrelievoLastra].Stato = INTERROTTO OR
					Programma_J[J_PosStartApproccioPrelLastra].Stato = INTERROTTO THEN
						Ciclo^.Passo := 90; 									
				ELSE
				//	IF BarcodeValido OR NOT HMI_AbilitaLettoreBC THEN //Valutazione dello stato di lettura del BC
						IF StepInto THEN
							Programma_Y[Y_PosPrelievoInLentaLastra].Stato 			:= DA_ESEGUIRE;
							Programma_Y[Y_PosPrelievoInLentaLastra].InterpolaAsse 	:= NO_INTERPOLAZIONE_ASSE;
							ProgrammaToModule_Y 									:= Programma_Y[Y_PosPrelievoInLentaLastra];
							//Sblocco pinza
							////TFParametersArrayClear(ADR(ParametersArray));
							////TFCommandSend(CmdSbloccaPinza,ParametersArray,Modules^.Pinza.Cmd);
							
							//IF NOT AttivazioneVuotoDistanza AND BarcodeValido THEN
							//	TFParametersArrayClear(ADR(ParametersArray));
							//	ParametersArray.Parameters[0] := BOOL_TO_STRING(NOT PrelievoPezzoOrizzontale);//SE TRUE: pezzo prelevato da cavallina, altrimenti prelievo orizzontale
							//	TFCommandSend(CmdPRELOAD,ParametersArray,Modules^.Pinza.Cmd);//LANCIO COMANDO ASPIRAZIONE PINZA
							//END_IF
							Ciclo^.Passo := 91;
							STEPDone := FALSE;
						END_IF
					//ELSE
					//	;
					//END_IF
				END_IF	
	
			(* Case 91 -  Attesa completamento dei comandi *)
			91: 
				IF Programma_Y[Y_PosPrelievoInLentaLastra].Stato = INTERROTTO OR 
					TFStateCodeGet(Modules^.Pinza.State) = StateERROR THEN
						Ciclo^.Passo := 91; 										
				ELSE
					IF (Programma_Y[Y_PosStartLentaPrelievoLastra].Stato = TERMINATO OR Asse_Y_InFinestraDiPassMode)then //AND
						//TFStateCodeGet(Modules^.Pinza.State) = StateSbloccaPinza_END THEN
						Ciclo^.Passo := 115;//100;
						STEPDone := FALSE;
					END_IF	
				END_IF
				
			(* Case 100 - Lancio Tasteggio J *)
			100:
				IF StepInto THEN
					HMI_AbilitaTasteggioRotazionePinza := false;
					IF HMI_AbilitaTasteggioRotazionePinza THEN
						Modules^.Ax_J.IN_Stop := FALSE;
						TFParametersArrayClear(ADR(ParametersArray));
						TFCommandSend(CmdTASTEGGIO,ParametersArray,Modules^.Ax_J.Cmd);//LANCIO COMANDO per tateggio inclinazione pinza
					END_IF
					//Ciclo^.Passo := 101;
					Ciclo^.Passo := 115;
					STEPDone := FALSE;
				END_IF

			(* Case 101 -  Attesa completamento del comando DI TASTEGGIO DELLA J*)
			101: 
				IF TFStateCodeGet(Modules^.AX_J.State) = StateError THEN
					Ciclo^.Passo := 101;																
				ELSE
					IF (TFStateCodeGet(Modules^.AX_J.State) >= StateTASTEGGIO_RUN + 10 AND TFStateCodeGet(Modules^.AX_J.State) <= StateTASTEGGIO_END) OR NOT HMI_AbilitaTasteggioRotazionePinza THEN		
						Ciclo^.Passo := 115;	
						STEPDone := TRUE;
					END_IF	
				END_IF
			
			(* Case 115 -  Attesa completamento del comando di tasteggio IN Y *)
			115: 
				IF TFStateCodeGet(Modules^.AX_J.State) = StateError OR 
					Programma_Y[Y_PosPrelievoInLentaLastra].Stato = INTERROTTO	THEN
						ReqStartAspirazione := FALSE;
						Ciclo^.Passo 		:= 115;																
				ELSE
					IF NOT ReqStartAspirazione AND AttivazioneVuotoDistanza THEN
						//IF Modules^.Pinza.OUT.DistanzaMedia <= 100 THEN
							ReqStartAspirazione := TRUE;
							TFParametersArrayClear(ADR(ParametersArray));
							ParametersArray.Parameters[0] := BOOL_TO_STRING(NOT PrelievoPezzoOrizzontale);// prelievo orizzontale
							ParametersArray.Parameters[1] := BOOL_TO_STRING(FALSE);//no falde
							TFCommandSend(CmdPRELOAD,ParametersArray,Modules^.Pinza.Cmd);//LANCIO COMANDO ASPIRAZIONE PINZA
						//END_IF
					END_IF
					IF Programma_Y[Y_PosPrelievoInLentaLastra].Stato = TERMINATO THEN//Pezzo in presa
						TFParametersArrayClear(ADR(ParametersArray));
						TFCommandSend(CmdCheckPresence,ParametersArray,Modules^.Pinza.Cmd);
						ReqStartAspirazione 	:= FALSE;
						Ciclo^.Passo 			:= 116;//dichiaro il ciclo terminato
						Modules^.Ax_J.IN_Stop 	:= TRUE; //Fermo Comando di tasteggio
						STEPDone 				:= TRUE;
						
					END_IF
				END_IF

			(* Case 116 - DISTACCO LASTRA *)
			116: 
				
				IF TFStateCodeGet(Modules^.Pinza.State) = StateCHECKPRESENCE_END AND  TFTimerDone(ADR(ReControlPiezaCogida)) THEN
					IF PinzaInPresa THEN
						IF StepInto THEN
							Programma_Z[Z_PosDistaccoLastraInLentaLastra].Stato 			:= DA_ESEGUIRE;
							Programma_Z[Z_PosDistaccoLastraInLentaLastra].InterpolaAsse 	:= INTERPOLAZIONE_ASSE;
							ProgrammaToModule_Z 											:= Programma_Z[Z_PosDistaccoLastraInLentaLastra];
	
							IF Modules^.AX_J.Ax^.Status.ActPosition > 90 THEN		
								Programma_Y[Y_PosDistaccoLastraInLentaLastra].Quota_Destinazione 	:= Modules^.AX_Y.QuotaAsseLetturaTasteggio + OffsetDistacco.Lastra.Y;
							ELSIF Modules^.AX_J.Ax^.Status.ActPosition < 90 THEN	
								Programma_Y[Y_PosDistaccoLastraInLentaLastra].Quota_Destinazione 	:= Modules^.AX_Y.QuotaAsseLetturaTasteggio - OffsetDistacco.Lastra.Y;
							END_IF
							Programma_Y[Y_PosDistaccoLastraInLentaLastra].Stato 			:= DA_ESEGUIRE;
							Programma_Y[Y_PosDistaccoLastraInLentaLastra].InterpolaAsse 	:= INTERPOLAZIONE_ASSE;
							ProgrammaToModule_Y 											:= Programma_Y[Y_PosDistaccoLastraInLentaLastra];
							
							HMI_AbilitaSfogliaturaJ := TRUE;
							HMI_GradiSfogliaturaJ := MIN(MAX(1,HMI_GradiSfogliaturaJ),3);
							IF HMI_AbilitaSfogliaturaJ THEN
								IF Modules^.AX_J.Ax^.Status.ActPosition > 90 THEN
									Programma_J[J_PosSfogliatura].Quota_Destinazione := MIN(180,Modules^.AX_J.Ax^.Status.ActPosition - HMI_GradiSfogliaturaJ);
								ELSIF Modules^.AX_J.Ax^.Status.ActPosition < 90 THEN
									Programma_J[J_PosSfogliatura].Quota_Destinazione := MAX(0,Modules^.AX_J.Ax^.Status.ActPosition + HMI_GradiSfogliaturaJ);
								END_IF
								Programma_J[J_PosSfogliatura].Stato 			 := DA_ESEGUIRE;
								//Programma_J[J_PosSfogliatura].InterpolaAsse 	 := INTERPOLAZIONE_ASSE;
								Programma_J[J_PosSfogliatura].InterpolaAsse 	 := No_INTERPOLAZIONE_ASSE;
								ProgrammaToModule_J 							 := Programma_J[J_PosSfogliatura];
							END_IF
			
							StartInterpolazioneAssi^ := TRUE; //Abilito l'interpolazione degli assi
							Ciclo^.Passo := 117;
							STEPDone := FALSE;
						END_IF	
					ELSE
						Errore := ErrMANCATO_PRELIEVO;
					END_IF
				ELSIF TFStateCodeGet(Modules^.Pinza.State) = StateERROR THEN
					Ciclo^.Passo := 116;
					Errore := ErrMalfunzionamentoSensoriPresenzaPinza;
				END_IF

			(* Case 117 -  Attesa completamento del comando *)
			117: 
				TimerPartenzaOk(IN:= Programma_Z[Z_PosDistaccoLastraInLentaLastra].Stato = TERMINATO AND 
								Programma_Y[Y_PosDistaccoLastraInLentaLastra].Stato = TERMINATO AND
								((Programma_J[J_PosSfogliatura].Stato = TERMINATO AND HMI_AbilitaSfogliaturaJ) OR NOT HMI_AbilitaSfogliaturaJ),
								PT:=TO_TIME(HMI_TempoAttesaPartenzaDopoPrelievo));//Setto un tempo di ritardo prima di partire...
				IF Programma_Z[Z_PosDistaccoLastraInLentaLastra].Stato = INTERROTTO OR
					Programma_Y[Y_PosDistaccoLastraInLentaLastra].Stato = INTERROTTO OR
					(Programma_J[J_PosSfogliatura].Stato = INTERROTTO AND HMI_AbilitaSfogliaturaJ) THEN
						Ciclo^.Passo := 117;																
				ELSE
					IF TimerPartenzaOk.Q THEN 
						//TFParametersArrayClear(ADR(ParametersArray));
						//TFCommandSend(CmdCheckPresence,ParametersArray,Modules^.Pinza.Cmd);
						Ciclo^.Passo := 118;//1000;//CICLO TERMINATO
					END_IF
				END_IF

			(* Case 118 -  Attesa completamento del comando *)
			118:
				IF PinzaInPresa THEN
						IF StepInto THEN
							Ciclo^.Passo := 1000;//CICLO TERMINATO
							Modules^.Ax_J.IN_Stop := TRUE; //Fermo Comando di tasteggio
							STEPDone := FALSE;
							SupportoVuoto := FALSE;
						END_IF
				ELSE//IF NOT Modules^.Pinza.StatoPinza.PianoInPresa THEN
					Ciclo^.Passo := 118;
					Errore := ErrMANCATO_PRELIEVO;
				END_IF

			(* Case 1000 *)
			1000:
				(* Stop tempo ciclo *)
				STEPDone := TRUE;
				Ciclo^.Stato := TERMINATO;
				Ciclo^.Passo := 1000;
				
			(* Case 9999 - Ciclo NON annullato o NON terminato*)
			9999:
				Ciclo^.Stato := INTERROTTO;
				Ciclo^.Passo := 9999;
	ELSE						
		;	
	END_CASE;
ELSE								//Se il ciclo deve essere interrotto, setto il suo nuovo stato
	Ciclo^.Stato := INTERROTTO;
END_IF
END_ACTION

END_FUNCTION_BLOCK

// ---- POUs/TFPalletizerDataTF/Utility Varie/TFAsseInFinestra.TcPOU
FUNCTION TFAsseInFinestra : bool //Valuta se l'asse è nella finsetra di posizione desiderata
VAR_INPUT
	Posizione_Attuale 	: LREAL;
	Posizione_Finale 	: LREAL;
	FinestraDiControllo : REAL;
END_VAR
VAR
END_VAR

TFAsseInFinestra := FALSE;

IF Posizione_Attuale >= (Posizione_Finale - FinestraDiControllo/2) AND Posizione_Attuale <= (Posizione_Finale + FinestraDiControllo/2) THEN
	TFAsseInFinestra := TRUE;
	RETURN;
END_IF

END_FUNCTION

// ---- POUs/TFCicliDiLavoro/Lastre/Cicli di Deposito Lastre/TFCiclo_Deposito_Lastra.TcPOU
FUNCTION_BLOCK TFCiclo_Deposito_Lastra
VAR_INPUT
	Ciclo 		: POINTER TO Stato_Ciclo_Lavoro;
	Programma 	: POINTER TO TFProgramma_Ciclo_Lastra;
	ModuleAX_X 	: POINTER TO TFModulePalletizer_Ax;
	ModuleAX_Y 	: POINTER TO TFModulePalletizer_Ax;
	ModuleAX_Z 	: POINTER TO TFModulePalletizer_Ax;
	ModuleAX_J 	: POINTER TO TFModulePalletizer_AxJ_Lastre;
	ModulePinza : POINTER TO TFModulePalletizer_Pinza;
	StartInterpolazioneAssi : POINTER TO BOOL;
	QuotaPassModePuntoIntermedio : ARRAY [1..3] OF REAL;
	AbilitazioneGlobalePassMode	: BOOL;
	InterrompiCiclo : BOOL;
	Abilita_Ciclo_Step : BOOL;
	Command_Step : BOOL;
	AbilitazioneAnticipoDinamicoMovimenti : BOOL;

END_VAR
VAR_OUTPUT
	STEPDone	: BOOL;
	Errore : UINT;
END_VAR
VAR
	ConAccostamentoZ : BOOL := FALSE;
	StepInto: BOOL;
	PinzaInPresa : BOOL;
	PinzaVerticale : BOOL;
END_VAR

(* Set della variabile che mi permette di fare lo STEP nel ciclo *)
TFTimerCall(ADR(ReMovEjeXCicloDeposito),TimeBase);
StepInto := (Abilita_Ciclo_Step AND Command_Step) OR NOT Abilita_Ciclo_Step;

(* Reset Anticipo Dinamico se non ho l'abilitazione *)
IF NOT AbilitazioneAnticipoDinamicoMovimenti OR NOT HMI_DisabilitaAnticipiGLOBALE THEN
	QuotaAnticipoDinamicaX_Raggiunta := FALSE;
	QuotaAnticipoDinamicaY_Raggiunta := FALSE;
	QuotaAnticipoDinamicaZ_Raggiunta := FALSE;
END_IF

PinzaInPresa 	:= ModulePinza^.StatoPinza.ElementoPrelevato AND  
					ModulePinza^.StatoPinza.LatoDxPiastrellaInPresa AND
					ModulePinza^.StatoPinza.LatoSxPiastrellaInPresa;

PinzaVerticale := NOT(ModuleAX_J^.Ax^.Status.ActPosition > 85 AND ModuleAX_J^.Ax^.Status.ActPosition < 95);

EjeYPosFueraIngombroCargado := TFAsseInFinestra(Posizione_Attuale :=  ModuleAX_Y^.Ax^.Status.ActPosition ,
 Posizione_Finale := Programma_Y[Y_PosFuoriIngombroVuotoLastra].Quota_Destinazione ,FinestraDiControllo := 30.0 );

EjeYPos0Ingombro :=  TFAsseInFinestra(Posizione_Attuale := ModuleAX_Y^.Ax^.Status.ActPosition ,
 Posizione_Finale := Programma_Y[Y_PosPasillo0grados].Quota_Destinazione ,FinestraDiControllo := 30.0 ) ;
 
EjeYPos180Ingombro := TFAsseInFinestra(Posizione_Attuale := ModuleAX_Y^.Ax^.Status.ActPosition ,
 Posizione_Finale := Programma_Y[Y_PosPasillo180grados].Quota_Destinazione ,FinestraDiControllo := 30.0 ) ;
 
 EjeyPosLentaCoger := TFAsseInFinestra(Posizione_Attuale := ModuleAX_Y^.Ax^.Status.ActPosition ,
 Posizione_Finale := Programma_Y[Y_PosStartLentaDepositoLastra].Quota_Destinazione ,FinestraDiControllo := 30.0 ) ;

IF Ciclo^.Passo = 27 THEN

TFTimerSet(ADR(ReMovEjeXCicloDeposito),1000, FALSE );	
ELSE
TFTimerSet(ADR(ReMovEjeX),1000, 
TFAsseInFinestra(Posizione_Attuale := ModuleAX_Y^.Ax^.Status.ActPosition ,
 Posizione_Finale := Programma_Y[Y_PosFuoriIngombroVuotoLastra].Quota_Destinazione ,FinestraDiControllo := 30.0 ) );	
END_IF
  Temp_Bool[69]:=TFAsseInFinestra (Posizione_Attuale := ModuleAX_Y^.Ax^.Status.ActPosition ,
 Posizione_Finale := Programma_Y[Y_PosFuoriIngombroVuotoLastra].Quota_Destinazione ,FinestraDiControllo := 30.0 );
IF NOT InterrompiCiclo THEN
	IF Ciclo^.Stato = TERMINATO OR Ciclo^.Stato = ANNULLATO THEN
		Ciclo^.Passo := 0;
	//ELSIF Ciclo^.Stato = INTERROTTO AND Ciclo^.Passo = 56 THEN
	//	Ciclo^.Passo := 56;
	ELSIF Ciclo^.Stato = INTERROTTO THEN//AND NOT Ciclo^.Passo = 56 THEN
		Ciclo^.Passo := 999;
	END_IF
	Ciclo^.Stato := IN_ESECUZIONE;
	CASE Ciclo^.Passo OF
			(* Case 0 *)
			0:  Ciclo^.Stato := IN_ESECUZIONE;
				Ciclo^.Passo := 10;
				Errore := 0;
				STEPDone := FALSE;
				
			(* Case 10 -  *)
			10:	MaterialeDepositatoSuLinea := FALSE;
				IF PinzaVerticale THEN
					Ciclo^.Passo := 25;
				ELSE
					Ciclo^.Passo := 20;
				END_IF
						
			(* Case 20 - PROGRAMMA[Z_PosFuoriIngombroCaricoLastra] ASSE Z -> TRASLAZIONE A QUOTA DI FUORI INGOMBRO CON lLASTRA A BORDO *)	
			20:	Ciclo^.Stato := IN_ESECUZIONE;
				IF StepInto THEN
					Programma_Z[Z_PosFuoriIngombroCaricoLastra].Stato 			:= DA_ESEGUIRE;
					Programma_Z[Z_PosFuoriIngombroCaricoLastra].InterpolaAsse 	:= NO_INTERPOLAZIONE_ASSE;
					ProgrammaToModule_Z 										:= Programma_Z[Z_PosFuoriIngombroCaricoLastra];
					Ciclo^.Passo := 21;
					STEPDone := FALSE;
				END_IF
				
			(* Case 21 - Attesa completamento del comando MOVETOPOS o del raggiungimento quota di Pre-Movimento se abilitata la funzione*)
			21: 
				IF Programma_Z[Z_PosFuoriIngombroCaricoLastra].Stato = INTERROTTO THEN
					Ciclo^.Passo := 21;		
				ELSIF Programma_Z[Z_PosFuoriIngombroCaricoLastra].Stato = TERMINATO OR
					Asse_Z_InFinestraDiPassMode THEN
					Ciclo^.Passo := 24; //
					STEPDone := TRUE;							
				END_IF
			
			(* Case 22 - Fuori ingombro J - NON usato in questa fase *)	
			22: IF Programma_Z[Z_PosFuoriIngombroCaricoLastra].Stato = INTERROTTO THEN
					 Ciclo^.Passo := 22;
				ELSIF Programma_Z[Z_PosFuoriIngombroCaricoLastra].Stato = TERMINATO OR 
						Asse_Z_InFinestraDiPassMode OR 
						QuotaAnticipoDinamicaZ_Raggiunta THEN
							IF StepInto AND Temp_Bool[3] THEN 
								Programma_J[J_PosFuoriIngombro].Stato 			:= DA_ESEGUIRE;
								Programma_J[J_PosFuoriIngombro].InterpolaAsse 	:= NO_INTERPOLAZIONE_ASSE;
								ProgrammaToModule_J		 						:= Programma_J[J_PosFuoriIngombro];
								Ciclo^.Passo := 23;
								STEPDone := FALSE;
							END_IF									
				END_IF
			
			(* Case 23 - Attesa completamento Fuori ingombro J *)	
			23: IF Programma_Z[Z_PosFuoriIngombroCaricoLastra].Stato = INTERROTTO OR 
					Programma_J[J_PosFuoriIngombro].Stato = INTERROTTO THEN
					 Ciclo^.Passo := 23;
				ELSIF (Programma_Z[Z_PosFuoriIngombroCaricoLastra].Stato = TERMINATO OR Asse_Z_InFinestraDiPassMode (*OR QuotaAnticipoDinamicaZ_Raggiunta*)) AND 
					(Programma_J[J_PosFuoriIngombro].Stato = TERMINATO OR Asse_J_InFinestraDiPassMode OR QuotaAnticipoDinamicaJ_Raggiunta) THEN
						Ciclo^.Passo := 24;
						STEPDone := TRUE;										
				END_IF	
							
				
			(* Case 24 - Scelgo in quale direzione devo muovermi per primo a seconda della disposizione delle postazioni *)	
			24:	
				IF Programma_Z[Z_PosFuoriIngombroCaricoLastra].Stato = INTERROTTO THEN
					Ciclo^.Passo := 21;	
				ELSE
					Ciclo^.Passo := 25;
				END_IF
					
		{Region "Dipsoizione postazioni lungo X"}		
			(* Case 25 - Vado a quota di fuori ingombro con Y e J *)
			25:	
						Temp_Bool[84] := ((WorkAreaState[PosRobot].Supporto.Tipologia = CAVALLETTO AND 
							workAreaState[Mission.PPlace].Supporto.Tipologia = BUNDLE)  OR MultiplesCavalletesReceta ) AND PosicionJOrigen <> PosicionJDestino  ;
					
				IF StepInto THEN
					IF PinzaVerticale THEN
						Programma_Z[Z_PosFuoriIngombroCaricoLastra].Stato 			:= DA_ESEGUIRE;
						Programma_Z[Z_PosFuoriIngombroCaricoLastra].InterpolaAsse 	:= INTERPOLAZIONE_ASSE;
						ProgrammaToModule_Z 										:= Programma_Z[Z_PosFuoriIngombroCaricoLastra];
					END_IF
					
					IF WorkAreaState[PosRobot].Supporto.Tipologia = BUNDLE  AND Programma_J[J_PosFuoriIngombro].Quota_Destinazione = 0 THEN
						(*
						//**********************************************************************
						Programma_Y[Y_PosPasillo0grados].Stato 				:= NON_ESEGUITO;
						Programma_Y[Y_PosPasillo180grados].Stato 			:= NON_ESEGUITO;
						Programma_Y[Y_PosFuoriIngombroCaricoLastra].Stato 	:= NON_ESEGUITO;
						//********************************************************************
						*)
  						Programma_Y[Y_PosgiroPieza].Stato 			:= DA_ESEGUIRE;
						Programma_Y[Y_PosgiroPieza].InterpolaAsse 	:= INTERPOLAZIONE_ASSE;
						ProgrammaToModule_Y 						:= Programma_Y[Y_PosgiroPieza];
						IF Temp_Bool[2] THEN 
							Ciclo^.Passo := 27;
							STEPDone := FALSE;
						END_IF
					ELSIF ((WorkAreaState[PosRobot].Supporto.Tipologia = CAVALLETTO AND 
							workAreaState[Mission.PPlace].Supporto.Tipologia = BUNDLE)  OR MultiplesCavalletesReceta ) AND  NuEstacionPiking <> 0  
								 THEN
							IF PosicionJActual = 0 THEN
								Programma_Y[Y_PosPasillo0grados].Stato 			:= DA_ESEGUIRE;
								Programma_Y[Y_PosPasillo0grados].InterpolaAsse 	:= INTERPOLAZIONE_ASSE;
								ProgrammaToModule_Y 							:= Programma_Y[Y_PosPasillo0grados];
								IF Temp_Bool[10] AND EjeYPos0Ingombro THEN 
									Ciclo^.Passo := 60;
									STEPDone := FALSE;
								END_IF
							END_IF
							IF PosicionJActual = 180  THEN
								Programma_Y[Y_PosPasillo180grados].Stato 			:= DA_ESEGUIRE;
								Programma_Y[Y_PosPasillo180grados].InterpolaAsse 	:= INTERPOLAZIONE_ASSE;
								ProgrammaToModule_Y 								:= Programma_Y[Y_PosPasillo180grados];
								IF Temp_Bool[10]AND EjeYPos180Ingombro THEN 
									Ciclo^.Passo := 60;
									STEPDone := FALSE;
								END_IF
							END_IF
							
							IF PosicionJActual = 90 THEN
								IF PosicionJDestino = 0 THEN
									Programma_Y[Y_PosPasillo0grados].Stato 			:= DA_ESEGUIRE;
									Programma_Y[Y_PosPasillo0grados].InterpolaAsse 	:= INTERPOLAZIONE_ASSE;
									ProgrammaToModule_Y 							:= Programma_Y[Y_PosPasillo0grados];
									
									Programma_J[Pos0TrasporteCavallete].Stato 						:= DA_ESEGUIRE;
									Programma_J[Pos0TrasporteCavallete].InterpolaAsse 				:= INTERPOLAZIONE_ASSE;
									ProgrammaToModule_J		 									:= Programma_J[Pos0TrasporteCavallete];
									
									IF Temp_Bool[10] AND EjeYPos0Ingombro THEN 
										Ciclo^.Passo := 60;
										STEPDone := FALSE;
									END_IF
								END_IF
								
								IF PosicionJDestino = 180  THEN
									Programma_Y[Y_PosPasillo180grados].Stato 			:= DA_ESEGUIRE;
									Programma_Y[Y_PosPasillo180grados].InterpolaAsse 	:= INTERPOLAZIONE_ASSE;
									ProgrammaToModule_Y 								:= Programma_Y[Y_PosPasillo180grados];
									
									Programma_J[Pos180TrasporteCavallete].Stato 						:= DA_ESEGUIRE;
									Programma_J[Pos180TrasporteCavallete].InterpolaAsse 				:= INTERPOLAZIONE_ASSE;
									ProgrammaToModule_J		 									:= Programma_J[Pos180TrasporteCavallete];
									
									IF Temp_Bool[10] AND EjeYPos180Ingombro THEN 
										Ciclo^.Passo := 60;
										STEPDone := FALSE;
									END_IF
								END_IF
								IF PosicionJDestino = 90  THEN//*************************************************
									Programma_Y[Y_PosFuoriIngombroCaricoLastra].Stato 			:= DA_ESEGUIRE;
									Programma_Y[Y_PosFuoriIngombroCaricoLastra].InterpolaAsse 	:= INTERPOLAZIONE_ASSE;
									ProgrammaToModule_Y 										:= Programma_Y[Y_PosFuoriIngombroCaricoLastra];
									
									
									Programma_J[J_PosFuoriIngombro].Stato 						:= DA_ESEGUIRE;
									Programma_J[J_PosFuoriIngombro].InterpolaAsse 				:= INTERPOLAZIONE_ASSE;
									ProgrammaToModule_J		 									:= Programma_J[J_PosFuoriIngombro];
									
									StartInterpolazioneAssi^ := TRUE; //Abilito l'interpolazione degli assi						
									IF Temp_Bool[90] THEN 
											Ciclo^.Passo := 26;
											STEPDone := FALSE;
									END_IF
								END_IF
							END_IF
						
					
						
							
					ELSIF (((WorkAreaState[PosRobot].Supporto.Tipologia = CAVALLETTO AND 
							workAreaState[Mission.PPlace].Supporto.Tipologia = BUNDLE ) OR MultiplesCavalletesReceta) AND PosicionJOrigen = PosicionJDestino ) OR 
								(WorkAreaState[PosRobot].Supporto.Tipologia = CASSA_STANDARD AND 	
								WorkAreaState[Mission.PPlace].Supporto.Tipologia = CASSA_STANDARD AND 
									PosicionJActual = PosicionJDestino ) 
								 												THEN
						(*
						//********************************************************************++
						Programma_Y[Y_PosPasillo0grados].Stato 				:= NON_ESEGUITO;
						Programma_Y[Y_PosPasillo180grados].Stato 			:= NON_ESEGUITO;
						Programma_Y[Y_PosgiroPieza].Stato 					:= NON_ESEGUITO;		 
						//********************************************************************++	
						*)	 
						Programma_Y[Y_PosFuoriIngombroCaricoLastra].Stato 			:= DA_ESEGUIRE;
						Programma_Y[Y_PosFuoriIngombroCaricoLastra].InterpolaAsse 	:= INTERPOLAZIONE_ASSE;
						ProgrammaToModule_Y 										:= Programma_Y[Y_PosFuoriIngombroCaricoLastra];
						
						
						Programma_J[J_PosFuoriIngombro].Stato 						:= DA_ESEGUIRE;
						Programma_J[J_PosFuoriIngombro].InterpolaAsse 				:= INTERPOLAZIONE_ASSE;
						ProgrammaToModule_J		 									:= Programma_J[J_PosFuoriIngombro];
						
						StartInterpolazioneAssi^ := TRUE; //Abilito l'interpolazione degli assi						
						IF Temp_Bool[90] THEN 
						Ciclo^.Passo := 26;
						STEPDone := FALSE;
						END_IF
					ELSIF workAreaState[PosRobot].Supporto.Tipologia = BUNDLE  AND  PosicionJOrigen = PosicionJDestino  
								 THEN
						(*
						//********************************************************************++
						Programma_Y[Y_PosPasillo0grados].Stato 				:= NON_ESEGUITO;
						Programma_Y[Y_PosPasillo180grados].Stato 			:= NON_ESEGUITO;
						Programma_Y[Y_PosgiroPieza].Stato 					:= NON_ESEGUITO;		 
						//********************************************************************++
						*)	
						Programma_Y[Y_PosFuoriIngombroCaricoLastra].Stato 			:= DA_ESEGUIRE;
						Programma_Y[Y_PosFuoriIngombroCaricoLastra].InterpolaAsse 	:= INTERPOLAZIONE_ASSE;
						ProgrammaToModule_Y 										:= Programma_Y[Y_PosFuoriIngombroCaricoLastra];
						
						
						Programma_J[J_PosFuoriIngombro].Stato 						:= DA_ESEGUIRE;
						Programma_J[J_PosFuoriIngombro].InterpolaAsse 				:= INTERPOLAZIONE_ASSE;
						ProgrammaToModule_J		 									:= Programma_J[J_PosFuoriIngombro];
						
						StartInterpolazioneAssi^ := TRUE; //Abilito l'interpolazione degli assi						
						IF Temp_Bool[90] THEN 
						Ciclo^.Passo := 26;
						STEPDone := FALSE;
						END_IF
					ELSE
						(*
						//********************************************************************++
						Programma_Y[Y_PosPasillo0grados].Stato 				:= NON_ESEGUITO;
						Programma_Y[Y_PosPasillo180grados].Stato 			:= NON_ESEGUITO;
						Programma_Y[Y_PosgiroPieza].Stato 					:= NON_ESEGUITO;		 
						//********************************************************************++
						*)	
						Programma_Y[Y_PosFuoriIngombroCaricoLastra].Stato 			:= DA_ESEGUIRE;
						Programma_Y[Y_PosFuoriIngombroCaricoLastra].InterpolaAsse 	:= INTERPOLAZIONE_ASSE;
						ProgrammaToModule_Y 										:= Programma_Y[Y_PosFuoriIngombroCaricoLastra];
						
						
						Programma_J[J_PosFuoriIngombro].Stato 						:= DA_ESEGUIRE;
						Programma_J[J_PosFuoriIngombro].InterpolaAsse 				:= INTERPOLAZIONE_ASSE;
						ProgrammaToModule_J		 									:= Programma_J[J_PosFuoriIngombro];
						
						StartInterpolazioneAssi^ := TRUE; //Abilito l'interpolazione degli assi						
						IF Temp_Bool[90] THEN 
						Ciclo^.Passo := 26;
						STEPDone := FALSE;
						END_IF
					END_IF 
					
				END_IF
					
					
				
			// VOY CON X A LA POSICION DE DEPOSITO
			60: 	IF 
 						(Programma_Y[Y_PosPasillo0grados].Stato 				= INTERROTTO AND PosicionJActual = 0) OR 
						(Programma_Y[Y_PosPasillo180grados].Stato 			= INTERROTTO AND PosicionJActual = 180 )OR 
						Programma_Z[Z_PosFuoriIngombroCaricoLastra].Stato 	= INTERROTTO OR 
						Programma_J[J_PosSfogliatura].Stato 				= INTERROTTO THEN
						Ciclo^.Passo := 60;
					ELSE	
						IF  ((Programma_Y[Y_PosPasillo0grados].Stato 				= TERMINATO AND PosicionJActual = 0) OR  
							(Programma_Y[Y_PosPasillo180grados].Stato 			= TERMINATO AND PosicionJActual = 180)) AND
							Programma_Z[Z_PosFuoriIngombroCaricoLastra].Stato 	= TERMINATO AND
							Programma_J[J_PosSfogliatura].Stato 				= TERMINATO THEN
								 	
							IF 	NOT MultiplesCavalletesReceta OR PosicionJDestino = 90 OR (WorkAreaState[Mission.PPlace].Supporto.Tipologia = BUNDLE AND MultiplesCavalletesReceta) THEN	
							Programma_X[X_PosStartLentaDepositoLastra].Stato 			:= DA_ESEGUIRE;
							Programma_X[X_PosStartLentaDepositoLastra].InterpolaAsse 	:= NO_INTERPOLAZIONE_ASSE;
							ProgrammaToModule_X 										:= Programma_X[X_PosStartLentaDepositoLastra];
							ELSE 
								Programma_X[X_PosGiroPiezaTraCavallete].Stato 			:= DA_ESEGUIRE;
								Programma_X[X_PosGiroPiezaTraCavallete].InterpolaAsse 	:= NO_INTERPOLAZIONE_ASSE;
								ProgrammaToModule_X 										:= Programma_X[X_PosGiroPiezaTraCavallete];
							END_IF
							IF Temp_Bool[11] THEN 
								Ciclo^.Passo := 61;
								STEPDone := FALSE;	
							END_IF
						END_IF 
					END_IF	
			 // VPY CON Y A LA POSICION DE GIRAR		
					
			61: 	IF (Programma_Y[Y_PosFuoriIngombroCaricoLastra].Stato 	= INTERROTTO AND ProgramaEjes.EjeY = 127)  OR 
						(Programma_Y[Y_PosPasillo0grados].Stato 				= INTERROTTO  AND  PosicionJActual = 0 AND ProgramaEjes.EjeY = 128 )OR
						(Programma_Y[Y_PosPasillo180grados].Stato 				= INTERROTTO  AND  PosicionJActual = 180 AND  ProgramaEjes.EjeY = 129)OR
						Programma_Z[Z_PosFuoriIngombroCaricoLastra].Stato 		= INTERROTTO OR 
						Programma_J[J_PosSfogliatura].Stato 					= INTERROTTO OR
						(Programma_X[X_PosStartLentaDepositoLastra].Stato 		= INTERROTTO AND ProgramaEjes.EjeX = 104) OR 
						(Programma_X[X_PosGiroPiezaTraCavallete].Stato 			= INTERROTTO AND  ProgramaEjes.EjeX = 127) 	THEN
						Ciclo^.Passo := 60;
					ELSE	
						IF ((Programma_Y[Y_PosFuoriIngombroCaricoLastra].Stato =  TERMINATO AND ProgramaEjes.EjeY = 127 )OR
							(Programma_Y[Y_PosPasillo0grados].Stato =  TERMINATO AND   PosicionJActual = 0 AND ProgramaEjes.EjeY = 128) OR
							(Programma_Y[Y_PosPasillo180grados].Stato =  TERMINATO AND  PosicionJActual = 180 AND ProgramaEjes.EjeY = 129 ))
							AND	Programma_Z[Z_PosFuoriIngombroCaricoLastra].Stato = TERMINATO 
								AND	Programma_J[J_PosSfogliatura].Stato = TERMINATO
									AND ((Programma_X[X_PosStartLentaDepositoLastra].Stato =TERMINATO AND ProgramaEjes.EjeX = 104) OR
									 (Programma_X[X_PosGiroPiezaTraCavallete].Stato =TERMINATO AND ProgramaEjes.EjeX = 127 )) AND PosicionJDestino <> 90 		THEN
									 
									 
								IF (Programma_X[X_PosGiroPiezaTraCavallete].Stato =TERMINATO AND ProgramaEjes.EjeX = 127) OR  
									(Programma_X[X_PosStartLentaDepositoLastra].Stato 		= TERMINATO AND ProgramaEjes.EjeX = 104 AND PosicionJActual <> PosicionJDestino)		THEN
									Programma_Y[Y_PosgiroPieza].Stato 			:= DA_ESEGUIRE;
									Programma_Y[Y_PosgiroPieza].InterpolaAsse 	:= INTERPOLAZIONE_ASSE;
									ProgrammaToModule_Y 						:= Programma_Y[Y_PosgiroPieza];
									IF Temp_Bool[12] THEN 
										Ciclo^.Passo := 62;
										STEPDone := FALSE;	
									END_IF
									ELSIF Programma_X[X_PosStartLentaDepositoLastra].Stato 		= TERMINATO AND ProgramaEjes.EjeX = 104 and PosicionJActual = PosicionJDestino THEN 
									IF Temp_Bool[12] THEN 
										Ciclo^.Passo := 31;
										STEPDone := FALSE;	
									END_IF	
								END_IF
							ELSIF  ((Programma_Y[Y_PosFuoriIngombroCaricoLastra].Stato =  TERMINATO AND ProgramaEjes.EjeY = 127 )OR
										(Programma_Y[Y_PosPasillo0grados].Stato =  TERMINATO AND   PosicionJActual = 0 AND ProgramaEjes.EjeY = 128) OR
											(Programma_Y[Y_PosPasillo180grados].Stato =  TERMINATO AND  PosicionJActual = 180 AND ProgramaEjes.EjeY = 129 ))
													AND	Programma_Z[Z_PosFuoriIngombroCaricoLastra].Stato = TERMINATO 
															AND	Programma_J[J_PosSfogliatura].Stato = TERMINATO
																AND ((Programma_X[X_PosStartLentaDepositoLastra].Stato =TERMINATO AND ProgramaEjes.EjeX = 104) OR
									 								(Programma_X[X_PosGiroPiezaTraCavallete].Stato =TERMINATO AND ProgramaEjes.EjeX = 127 )) AND PosicionJDestino = 90	 THEN 
										IF Temp_Bool[12] THEN 
										Ciclo^.Passo := 31;
										STEPDone := FALSE;	
									END_IF						
						END_IF 
					END_IF	
			62: 	IF Programma_Y[Y_PosgiroPieza].Stato 	= INTERROTTO  OR 
						Programma_Z[Z_PosFuoriIngombroCaricoLastra].Stato 	= INTERROTTO OR 
						Programma_J[J_PosSfogliatura].Stato 				= INTERROTTO OR
						Programma_X[X_PosStartLentaDepositoLastra].Stato 	= INTERROTTO AND NOT MultiplesCavalletesReceta OR 
						Programma_X[X_PosGiroPiezaTraCavallete].Stato 	= INTERROTTO AND MultiplesCavalletesReceta	 THEN
						Ciclo^.Passo := 62;
					ELSE	
						IF Programma_Y[Y_PosgiroPieza].Stato =  TERMINATO 	
								AND	Programma_Z[Z_PosFuoriIngombroCaricoLastra].Stato = TERMINATO 
									AND	Programma_J[J_PosSfogliatura].Stato = TERMINATO
									AND Programma_X[X_PosStartLentaDepositoLastra].Stato =TERMINATO AND NOT MultiplesCavalletesReceta OR 	
										Programma_X[X_PosGiroPiezaTraCavallete].Stato =TERMINATO AND  MultiplesCavalletesReceta	THEN
							Programma_J[J_PosFuoriIngombro].Stato 						:= DA_ESEGUIRE;
							Programma_J[J_PosFuoriIngombro].InterpolaAsse 				:= INTERPOLAZIONE_ASSE;
							ProgrammaToModule_J		 									:= Programma_J[J_PosFuoriIngombro];
							IF Temp_Bool[13] THEN 
								Ciclo^.Passo := 63;
								STEPDone := FALSE;	
							END_IF
						END_IF 
					END_IF	
			63: 	IF Programma_Y[Y_PosgiroPieza].Stato 	= INTERROTTO  OR 
						Programma_Z[Z_PosFuoriIngombroCaricoLastra].Stato 	= INTERROTTO OR 
						Programma_J[J_PosFuoriIngombro].Stato 				= INTERROTTO OR
						Programma_X[X_PosStartLentaDepositoLastra].Stato 	= INTERROTTO AND NOT MultiplesCavalletesReceta OR
						Programma_X[X_PosGiroPiezaTraCavallete].Stato =INTERROTTO AND  MultiplesCavalletesReceta THEN
						Ciclo^.Passo := 63;
					ELSE	
						IF Programma_Y[Y_PosgiroPieza].Stato =  TERMINATO 	
								AND	Programma_Z[Z_PosFuoriIngombroCaricoLastra].Stato = TERMINATO 
									AND	Programma_J[J_PosFuoriIngombro].Stato = TERMINATO
									AND (Programma_X[X_PosStartLentaDepositoLastra].Stato =TERMINATO AND NOT MultiplesCavalletesReceta) OR
									(Programma_X[X_PosGiroPiezaTraCavallete].Stato = TERMINATO AND  MultiplesCavalletesReceta )	THEN
						(*
						//********************************************************************++
						Programma_Y[Y_PosPasillo0grados].Stato 				:= NON_ESEGUITO;
						Programma_Y[Y_PosPasillo180grados].Stato 			:= NON_ESEGUITO;
						Programma_Y[Y_PosgiroPieza].Stato 					:= NON_ESEGUITO;		 
						//********************************************************************++
						*)	
							Programma_Y[Y_PosFuoriIngombroCaricoLastra].Stato 			:= DA_ESEGUIRE;
							Programma_Y[Y_PosFuoriIngombroCaricoLastra].InterpolaAsse 	:= INTERPOLAZIONE_ASSE;
							ProgrammaToModule_Y 										:= Programma_Y[Y_PosFuoriIngombroCaricoLastra];
							IF Temp_Bool[14] THEN 
								Ciclo^.Passo := 64;
								STEPDone := FALSE;	
							END_IF
						END_IF 
					END_IF	
			64 :
				 IF Programma_X[X_PosStartLentaDepositoLastra].Stato = INTERROTTO AND NOT MultiplesCavalletesReceta OR
					Programma_X[X_PosGiroPiezaTraCavallete].Stato = INTERROTTO AND  MultiplesCavalletesReceta OR 
					Programma_Y[Y_PosFuoriIngombroCaricoLastra].Stato = INTERROTTO OR
					Programma_Z[Z_PosFuoriIngombroCaricoLastra].Stato = INTERROTTO OR 
					Programma_J[J_PosFuoriIngombro].Stato = INTERROTTO THEN
						Ciclo^.Passo := 64;
				ELSE	
						IF (Programma_Y[Y_PosFuoriIngombroCaricoLastra].Stato =  TERMINATO AND ProgramaEjes.EjeY = 126) AND 	
							Programma_Z[Z_PosFuoriIngombroCaricoLastra].Stato = TERMINATO AND
							Programma_J[J_PosFuoriIngombro].Stato = TERMINATO AND 
									((Programma_X[X_PosStartLentaDepositoLastra].Stato =TERMINATO AND NOT MultiplesCavalletesReceta) OR
									(Programma_X[X_PosGiroPiezaTraCavallete].Stato = TERMINATO AND  MultiplesCavalletesReceta ) )AND  Temp_Bool[69] AND  Temp_Bool[70]	THEN
							Programma_X[X_PosStartLentaDepositoLastra].Stato 			:= DA_ESEGUIRE;
							Programma_X[X_PosStartLentaDepositoLastra].InterpolaAsse 	:= NO_INTERPOLAZIONE_ASSE;
							ProgrammaToModule_X 										:= Programma_X[X_PosStartLentaDepositoLastra];
							IF Temp_Bool[18] THEN 
								Ciclo^.Passo := 31;
								STEPDone := FALSE;	
							END_IF
						END_IF 
				END_IF	
			
					
			27: 	IF Programma_Y[Y_PosgiroPieza].Stato 	= INTERROTTO  OR 
						Programma_Z[Z_PosFuoriIngombroCaricoLastra].Stato 	= INTERROTTO OR 
						Programma_J[J_PosFuoriIngombro].Stato 				= INTERROTTO THEN
						Ciclo^.Passo := 27;
					ELSE	
						IF Programma_Y[Y_PosgiroPieza].Stato =  TERMINATO 		THEN
							Programma_J[J_PosFuoriIngombro].Stato 						:= DA_ESEGUIRE;
							Programma_J[J_PosFuoriIngombro].InterpolaAsse 				:= No_INTERPOLAZIONE_ASSE;
							ProgrammaToModule_J		 									:= Programma_J[J_PosFuoriIngombro];
							IF Temp_Bool[11] THEN 
							Ciclo^.Passo := 28;
							STEPDone := FALSE;	
					END_IF
						END_IF 
					END_IF
					
			28: 	IF Programma_Y[Y_PosgiroPieza].Stato 	= INTERROTTO  OR 
						Programma_Z[Z_PosFuoriIngombroCaricoLastra].Stato 	= INTERROTTO OR 
						Programma_J[J_PosFuoriIngombro].Stato 				= INTERROTTO THEN
						Ciclo^.Passo := 27;
					ELSE	
						IF Programma_Y[Y_PosgiroPieza].Stato =  TERMINATO AND Programma_J[J_PosFuoriIngombro].Stato = TERMINATO	 	THEN
							
						(*
						//********************************************************************++
						Programma_Y[Y_PosPasillo0grados].Stato 				:= NON_ESEGUITO;
						Programma_Y[Y_PosPasillo180grados].Stato 			:= NON_ESEGUITO;
						Programma_Y[Y_PosgiroPieza].Stato 					:= NON_ESEGUITO;		 
						//********************************************************************++
						*)	
							Programma_Y[Y_PosFuoriIngombroCaricoLastra].Stato 			:= DA_ESEGUIRE;
							Programma_Y[Y_PosFuoriIngombroCaricoLastra].InterpolaAsse 	:= INTERPOLAZIONE_ASSE;
							ProgrammaToModule_Y 										:= Programma_Y[Y_PosFuoriIngombroCaricoLastra];
							IF Temp_Bool[12] THEN 
							Ciclo^.Passo := 26;
							STEPDone := FALSE;	
							END_IF
						END_IF 
					END_IF
					
			(* Case 26 - Check se a quota di fuori ingombro con Y & J *)		
			26:	IF Programma_Y[Y_PosFuoriIngombroCaricoLastra].Stato 	= INTERROTTO OR 
					Programma_Z[Z_PosFuoriIngombroCaricoLastra].Stato 	= INTERROTTO OR 
					Programma_J[J_PosFuoriIngombro].Stato 				= INTERROTTO THEN
						Ciclo^.Passo := 26;
				ELSE	
				IF WorkAreaState[PosRobot].Supporto.Tipologia = BUNDLE  AND Programma_J[J_PosFuoriIngombro].Quota_Destinazione = 0 THEN
					IF  Programma_Y[Y_PosFuoriIngombroCaricoLastra].Stato = TERMINATO  AND
						Programma_J[J_PosFuoriIngombro].Stato = TERMINATO  AND
						Programma_Z[Z_PosFuoriIngombroCaricoLastra].Stato = TERMINATO THEN
						IF Temp_Bool[91] THEN 
						Ciclo^.Passo := 30;
						STEPDone := TRUE;	
						END_IF						
					END_IF
				ELSE
					IF (Programma_Y[Y_PosFuoriIngombroCaricoLastra].Stato = TERMINATO OR Asse_Y_InFinestraDiPassMode OR QuotaAnticipoDinamicaY_Raggiunta) AND
						(Programma_J[J_PosFuoriIngombro].Stato = TERMINATO OR Asse_J_InFinestraDiPassMode OR QuotaAnticipoDinamicaJ_Raggiunta) AND
						Programma_Z[Z_PosFuoriIngombroCaricoLastra].Stato = TERMINATO THEN
						IF Temp_Bool[92] THEN 
						Ciclo^.Passo := 30;
						STEPDone := TRUE;	
						END_IF
					END_IF
				END_IF	
				END_IF
										
			(* Case 30 - PROGRAMMA[0] ASSE X  -> TRASLAZIONE A QUOTA DI DEPOSITO  *)	
			30:	IF Programma_Z[Z_PosFuoriIngombroCaricoLastra].Stato = INTERROTTO OR 
					Programma_Y[Y_PosFuoriIngombroCaricoLastra].Stato = INTERROTTO OR 
					Programma_J[J_PosFuoriIngombro].Stato = INTERROTTO THEN
						Ciclo^.Passo := 30;										
				ELSE
					IF StepInto THEN
						Programma_X[X_PosStartLentaDepositoLastra].Stato 			:= DA_ESEGUIRE;
						Programma_X[X_PosStartLentaDepositoLastra].InterpolaAsse 	:= NO_INTERPOLAZIONE_ASSE;
						ProgrammaToModule_X 										:= Programma_X[X_PosStartLentaDepositoLastra];
						IF Temp_Bool[93] THEN 
						Ciclo^.Passo := 31;
						STEPDone := FALSE;
						END_IF
					END_IF
				END_IF			
			
			(* Case 31 -  Attesa completamento del comando MOVETOPOS o del raggiungimento quota di Pre-Movimento se abilitata la funzione *)
			31: 
				IF Programma_X[X_PosStartLentaDepositoLastra].Stato = INTERROTTO   OR
					(Programma_Y[Y_PosFuoriIngombroCaricoLastra].Stato = INTERROTTO AND  ProgramaEjes.EjeY = 104 ) OR
					(Programma_Y[Y_PosPasillo0grados].Stato = INTERROTTO AND  ProgramaEjes.EjeY = 128)  OR
					(Programma_Y[Y_PosPasillo180grados].Stato = INTERROTTO AND  ProgramaEjes.EjeY = 129)  OR
					Programma_Z[Z_PosFuoriIngombroCaricoLastra].Stato = INTERROTTO OR 
					Programma_J[J_PosFuoriIngombro].Stato = INTERROTTO THEN
						Ciclo^.Passo := 31;
				ELSE	
					IF (Programma_X[X_PosStartLentaDepositoLastra].Stato = TERMINATO OR Asse_X_InFinestraDiPassMode OR QuotaAnticipoDinamicaX_Raggiunta) THEN 
						IF WorkAreaState[Mission.PPlace].Supporto.Tipologia <> CAVALLETTO AND WorkAreaState[Mission.PPlace].Supporto.Tipologia <> BUNDLE THEN //se non devo depositare nel cavalletto...	
							Ciclo^.Passo := 32;//ciclo per orizzontale
						ELSE
							Ciclo^.Passo := 40;//Ciclo per cavalletto
						END_IF
						STEPDone := TRUE;							
					END_IF
				END_IF
				
			(* Case 32 - Vado a quota di START LENTA CON GLI ASSI con Y,Z,J *)
			32:
				IF Programma_X[X_PosStartLentaDepositoLastra].Stato = INTERROTTO OR
					(Programma_Y[Y_PosFuoriIngombroCaricoLastra].Stato = INTERROTTO AND  ProgramaEjes.EjeY = 104 ) OR
					(Programma_Y[Y_PosPasillo0grados].Stato = INTERROTTO AND  ProgramaEjes.EjeY = 128)  OR
					(Programma_Y[Y_PosPasillo180grados].Stato = INTERROTTO AND  ProgramaEjes.EjeY = 129)  OR
					Programma_Z[Z_PosFuoriIngombroCaricoLastra].Stato = INTERROTTO OR 
					Programma_J[J_PosFuoriIngombro].Stato = INTERROTTO THEN
						Ciclo^.Passo := 32;										
				ELSE
					IF StepInto AND Programma_X[X_PosStartLentaDepositoLastra].Stato = TERMINATO  THEN
						TFParametersArrayClear(ADR(ParametersArray));
						Programma_Y[Y_PosStartLentaDepositoLastra].Stato 			:= DA_ESEGUIRE;
						Programma_Y[Y_PosStartLentaDepositoLastra].InterpolaAsse 	:= INTERPOLAZIONE_ASSE;
						ProgrammaToModule_Y 										:= Programma_Y[Y_PosStartLentaDepositoLastra];
				
						//Programma_Z[Z_PosStartLentaDepositoLastra].Stato 			:= DA_ESEGUIRE;
						//Programma_Z[Z_PosStartLentaDepositoLastra].InterpolaAsse 	:= INTERPOLAZIONE_ASSE;
						//ProgrammaToModule_Z 										:= Programma_Z[Z_PosStartLentaDepositoLastra];
						
						Programma_J[J_PosDepositoLastra].Stato 						:= DA_ESEGUIRE;
						Programma_J[J_PosDepositoLastra].InterpolaAsse 				:= INTERPOLAZIONE_ASSE;
						ProgrammaToModule_J 										:= Programma_J[J_PosDepositoLastra];
						
						StartInterpolazioneAssi^ := TRUE; //Abilito l'interpolazione degli assi
												
						Ciclo^.Passo := 33;
						STEPDone := FALSE;
					END_IF
				END_IF
			
			(* Case 33 - Attendo completamento comando o assi in finsetra *)
			33:
				IF Programma_Y[Y_PosStartLentaDepositoLastra].Stato 	= TERMINATO OR ((Asse_Y_InFinestraDiPassMode OR TRUE) AND WorkAreaState[Mission.PPlace].Supporto.Tipologia <> CAVALLETTO AND WorkAreaState[Mission.PPlace].Supporto.Tipologia <> BUNDLE) AND 
					Programma_J[J_PosDepositoLastra].Stato 				= TERMINATO OR ((Asse_J_InFinestraDiPassMode OR TRUE) AND WorkAreaState[Mission.PPlace].Supporto.Tipologia <> CAVALLETTO AND WorkAreaState[Mission.PPlace].Supporto.Tipologia <> BUNDLE) AND
					Programma_X[X_PosStartLentaDepositoLastra].Stato 	= TERMINATO (*OR Asse_X_InFinestraDiPassMode)*)THEN// AND 
					//Programma_Z[Z_PosStartLentaDepositoLastra].Stato 	= TERMINATO (*OR Asse_Z_InFinestraDiPassMode)*) THEN
					IF EjeyPosLentaCoger THEN
						Programma_Z[Z_PosStartLentaDepositoLastra].Stato 			:= DA_ESEGUIRE;
						Programma_Z[Z_PosStartLentaDepositoLastra].InterpolaAsse 	:= NO_INTERPOLAZIONE_ASSE;
						ProgrammaToModule_Z 										:= Programma_Z[Z_PosStartLentaDepositoLastra];			

						Ciclo^.Passo := 34;
						STEPDone := TRUE;
					END_IF
						
				ELSIF Programma_Y[Y_PosStartLentaDepositoLastra].Stato 	= INTERROTTO OR 
					Programma_J[J_PosDepositoLastra].Stato 				= INTERROTTO OR 
					Programma_X[X_PosStartLentaDepositoLastra].Stato 	= INTERROTTO THEN//OR
				//	Programma_Z[Z_PosStartLentaDepositoLastra].Stato 	= TERMINATO THEN
						Ciclo^.Passo := 33;								
				END_IF

			(* Case 34 - Vado a quota di finale con Z *)
			34:
				IF Programma_X[X_PosStartLentaDepositoLastra].Stato = INTERROTTO OR
					Programma_Y[Y_PosStartLentaDepositoLastra].Stato = INTERROTTO OR
					Programma_J[J_PosDepositoLastra].Stato = INTERROTTO OR 
					Programma_Z[Z_PosStartLentaDepositoLastra].Stato 	= INTERROTTO THEN
						Ciclo^.Passo := 34;										
				ELSE
					IF Programma_Z[Z_PosStartLentaDepositoLastra].Stato 	= TERMINATO THEN
						IF StepInto THEN
							TFParametersArrayClear(ADR(ParametersArray));
							//Programma_Y[Y_PosDepositoInLentaLastra].Stato 			:= DA_ESEGUIRE;
							//Programma_Y[Y_PosDepositoInLentaLastra].InterpolaAsse 	:= INTERPOLAZIONE_ASSE;
							//ProgrammaToModule_Y 									:= Programma_Y[Y_PosDepositoInLentaLastra];
					
							Programma_Z[Z_PosDepositoInLentaLastra].Stato 			:= DA_ESEGUIRE;
							Programma_Z[Z_PosDepositoInLentaLastra].InterpolaAsse 	:= NO_INTERPOLAZIONE_ASSE;
							ProgrammaToModule_Z 									:= Programma_Z[Z_PosDepositoInLentaLastra];
													
							StartInterpolazioneAssi^ := TRUE; //Abilito l'interpolazione degli assi
													
							Ciclo^.Passo := 35;
							STEPDone := FALSE;
						END_IF
					END_IF
				END_IF

			(* Case 35 - Attendo completamento comando o assi in finsetra *)
			35:
				IF 	Programma_Z[Z_PosDepositoInLentaLastra].Stato = TERMINATO (*OR Asse_Z_InFinestraDiPassMode)*) THEN
					Ciclo^.Passo := 90;
					STEPDone := TRUE;
				ELSIF Programma_Z[Z_PosDepositoInLentaLastra].Stato = INTERROTTO THEN
					Ciclo^.Passo := 35;								
				END_IF
		{endregion}

		{Region "CICLO CAVALLETTO"}							
			(* Case 40 - Vado a quota di START LENTA CON GLI ASSI con Y,Z *)
			40:
				IF Programma_X[X_PosStartLentaDepositoLastra].Stato = INTERROTTO OR
					Programma_Y[Y_PosFuoriIngombroCaricoLastra].Stato = INTERROTTO OR
					Programma_Z[Z_PosFuoriIngombroCaricoLastra].Stato = INTERROTTO OR 
					Programma_J[J_PosFuoriIngombro].Stato = INTERROTTO THEN
						Ciclo^.Passo := 40;										
				ELSE
					IF StepInto THEN
						TFParametersArrayClear(ADR(ParametersArray));
						Programma_Y[Y_PosStartLentaDepositoLastra].Stato 			:= DA_ESEGUIRE;
						Programma_Y[Y_PosStartLentaDepositoLastra].InterpolaAsse 	:= INTERPOLAZIONE_ASSE;
						ProgrammaToModule_Y 										:= Programma_Y[Y_PosStartLentaDepositoLastra];
				
						Programma_Z[Z_PosStartLentaDepositoLastra].Stato 			:= DA_ESEGUIRE;
						Programma_Z[Z_PosStartLentaDepositoLastra].InterpolaAsse 	:= INTERPOLAZIONE_ASSE;
						ProgrammaToModule_Z 										:= Programma_Z[Z_PosStartLentaDepositoLastra];
						
						Programma_J[J_PosDepositoLastra].Quota_Destinazione    		:= Programma_J[J_PosDepositoLastra].Quota_Destinazione;
						Programma_J[J_PosDepositoLastra].Stato 						:= DA_ESEGUIRE;
						Programma_J[J_PosDepositoLastra].InterpolaAsse 				:= NO_INTERPOLAZIONE_ASSE;
						ProgrammaToModule_J 										:= Programma_J[J_PosDepositoLastra];
						
						StartInterpolazioneAssi^ := TRUE; //Abilito l'interpolazione degli assi
												
						Ciclo^.Passo := 41;
						STEPDone := FALSE;
					END_IF
				END_IF
			
			(* Case 41 - Vado a quota di finale con Z *)
			41:
				

				IF Programma_X[X_PosStartLentaDepositoLastra].Stato = INTERROTTO OR
					Programma_Y[Y_PosStartLentaDepositoLastra].Stato = INTERROTTO OR
					Programma_J[J_PosDepositoLastra].Stato = INTERROTTO OR 
					Programma_Z[Z_PosStartLentaDepositoLastra].Stato 	= INTERROTTO THEN
						Ciclo^.Passo := 41;										
				ELSE
					IF Programma_Y[Y_PosStartLentaDepositoLastra].Stato = TERMINATO  AND
						Programma_J[J_PosDepositoLastra].Stato = TERMINATO AND
						Programma_Z[Z_PosStartLentaDepositoLastra].Stato = TERMINATO AND NOT STEPDone THEN
							STEPDone := TRUE;
					ELSIF STEPDone THEN 	
							IF StepInto THEN
								TFParametersArrayClear(ADR(ParametersArray));
								Programma_Y[Y_PosDepositoInLentaLastra].Stato 			:= DA_ESEGUIRE;
								Programma_Y[Y_PosDepositoInLentaLastra].InterpolaAsse 	:= INTERPOLAZIONE_ASSE;
								ProgrammaToModule_Y 									:= Programma_Y[Y_PosDepositoInLentaLastra];
						
								Programma_Z[Z_PosDepositoInLentaLastra].Stato 			:= DA_ESEGUIRE;
								Programma_Z[Z_PosDepositoInLentaLastra].InterpolaAsse 	:= INTERPOLAZIONE_ASSE;
								ProgrammaToModule_Z 									:= Programma_Z[Z_PosDepositoInLentaLastra];
														
								StartInterpolazioneAssi^ := TRUE; //Abilito l'interpolazione degli assi
														
								Ciclo^.Passo := 42;
								STEPDone := FALSE;
							END_IF
					END_IF
				END_IF
			
			(* Case 42 - Attesa completamento posizionamento di tutti gli assi e stacco aspirazione *)
			42: 
				IF Programma_X[X_PosStartLentaDepositoLastra].Stato = INTERROTTO OR
					Programma_Y[Y_PosDepositoInLentaLastra].Stato = INTERROTTO OR
					Programma_Z[Z_PosDepositoInLentaLastra].Stato 	= INTERROTTO THEN
						Ciclo^.Passo := 42;										
				ELSE
					IF Programma_Y[Y_PosDepositoInLentaLastra].Stato = TERMINATO AND
						Programma_Z[Z_PosDepositoInLentaLastra].Stato = TERMINATO AND NOT STEPDone THEN
						 STEPDone:= TRUE;
					ELSIF STEPDone THEN	
						IF StepInto THEN
							TFParametersArrayClear(ADR(ParametersArray));
							TFCommandSend(CmdUNLOAD,ParametersArray,ModulePinza^.Cmd);
							Ciclo^.Passo := 43;
							STEPDone := FALSE;
						END_IF	
					END_IF						
				END_IF

			(* Case 43 - Attesa completamento rilascio pezzo *)	
			43:
				IF TFStateCodeGet(ModulePinza^.State) = StateError THEN
					Ciclo^.Passo := 43;																
				ELSE
					STEPDone := TRUE;
					IF TFStateCodeGet(ModulePinza^.State) = StateUNLOAD_END THEN//Pezzo rilasciato
						Ciclo^.Passo := 45;//
					END_IF	
				END_IF

			(* Case 44 - Vado a quota di finale con J *)
			44:
				IF Programma_X[X_PosStartLentaDepositoLastra].Stato = INTERROTTO OR
					Programma_Y[Y_PosDepositoInLentaLastra].Stato = INTERROTTO OR
					Programma_Z[Z_PosDepositoInLentaLastra].Stato 	= INTERROTTO THEN
						Ciclo^.Passo := 44;										
				ELSE
					IF Programma_Y[Y_PosDepositoInLentaLastra].Stato = TERMINATO AND
						Programma_Z[Z_PosDepositoInLentaLastra].Stato = TERMINATO THEN
							IF StepInto THEN
								TFParametersArrayClear(ADR(ParametersArray));
								Programma_J[J_PosDepositoLastra].Stato 						:= DA_ESEGUIRE;
								Programma_J[J_PosDepositoLastra].InterpolaAsse 				:= NO_INTERPOLAZIONE_ASSE;
								ProgrammaToModule_J 										:= Programma_J[J_PosDepositoLastra];
								Ciclo^.Passo := 45;
								STEPDone := FALSE;
							END_IF
					END_IF
				END_IF

			(* Case 45 - Attendo completamento comando o assi in finsetra *)
			45:
				//IF Programma_J[J_PosDepositoLastra].Stato = TERMINATO THEN
				IF StepInto THEN	
					//********************************************************************++
						Programma_Y[Y_PosPasillo0grados].Stato 				:= NON_ESEGUITO;
						Programma_Y[Y_PosPasillo180grados].Stato 			:= NON_ESEGUITO;
						Programma_Y[Y_PosgiroPieza].Stato 					:= NON_ESEGUITO;		 
						//********************************************************************++	
				
					Programma_Y[Y_PosFuoriIngombroCaricoLastra].Stato 			:= DA_ESEGUIRE;
					Programma_Y[Y_PosFuoriIngombroCaricoLastra].InterpolaAsse 	:= NO_INTERPOLAZIONE_ASSE;
					ProgrammaToModule_Y 										:= Programma_Y[Y_PosFuoriIngombroCaricoLastra];
			
					Programma_Z[Z_PosFuoriIngombroCaricoLastra].Stato 			:= DA_ESEGUIRE;
					Programma_Z[Z_PosFuoriIngombroCaricoLastra].InterpolaAsse 	:= NO_INTERPOLAZIONE_ASSE;
					ProgrammaToModule_Z 										:= Programma_Z[Z_PosFuoriIngombroCaricoLastra];
				
					//Programma_J[J_PosFuoriIngombro].Stato 						:= DA_ESEGUIRE;
					//Programma_J[J_PosFuoriIngombro].InterpolaAsse 				:= INTERPOLAZIONE_ASSE;
					//ProgrammaToModule_J		 									:= Programma_J[J_PosFuoriIngombro];
					Ciclo^.Passo := 46;	
					STEPDone := FALSE;
				END_IF
				//ELSIF Programma_J[J_PosDepositoLastra].Stato = INTERROTTO THEN
				//	Ciclo^.Passo := 45;								
				//END_IF	

			(* Case 46 - Attendo completamento comando o assi in finsetra *)
			46:
				IF Programma_Z[Z_PosFuoriIngombroCaricoLastra].Stato = TERMINATO AND 
					Programma_Y[Y_PosFuoriIngombroCaricoLastra].Stato = TERMINATO THEN//AND
					//Programma_J[J_PosFuoriIngombro].Stato = TERMINATO THEN
						Ciclo^.Passo := 1000;	
						STEPDone := TRUE;
				ELSIF Programma_Z[Z_PosFuoriIngombroCaricoLastra].Stato = INTERROTTO AND  
					  Programma_Y[Y_PosFuoriIngombroCaricoLastra].Stato = INTERROTTO THEN
					Ciclo^.Passo := 46;								
				END_IF	
		{endregion}


		{Region "Dipsoizione postazioni lungo Y"}							
			(* Case 50 - Vado a quota di deposito con X *)
			50:	IF Programma_Z[Z_PosFuoriIngombroCaricoLastra].Stato = INTERROTTO OR
					Programma_J[J_PosFuoriIngombro].Stato = INTERROTTO THEN
						Ciclo^.Passo := 50;										
				ELSE
					IF StepInto THEN
						Programma_X[X_PosStartLentaDepositoLastra].Stato 			:= DA_ESEGUIRE;
						Programma_X[X_PosStartLentaDepositoLastra].InterpolaAsse 	:= NO_INTERPOLAZIONE_ASSE;
						ProgrammaToModule_X 										:= Programma_X[X_PosStartLentaDepositoLastra];
						Ciclo^.Passo := 51;
						STEPDone := FALSE;
					END_IF
				END_IF
					
			(* Case 51 - Check se a quota di deposito X *)		
			51:	IF Programma_X[X_PosStartLentaDepositoLastra].Stato = INTERROTTO OR 
					Programma_Z[Z_PosFuoriIngombroCaricoLastra].Stato = INTERROTTO OR 
					Programma_J[J_PosFuoriIngombro].Stato = INTERROTTO THEN
						Ciclo^.Passo := 51;
				ELSE	
					IF Programma_X[X_PosStartLentaDepositoLastra].Stato = TERMINATO OR 
						Asse_X_InFinestraDiPassMode THEN
							Ciclo^.Passo := 52;
							STEPDone := TRUE;							
					END_IF
				END_IF
										
			(* Case 52 - lancio posizionamento Y,j e x se non serve fuori ingombro  *)	
			52:	IF Programma_Z[Z_PosFuoriIngombroCaricoLastra].Stato = INTERROTTO OR 
					(Programma_X[X_PosStartLentaDepositoLastra].Stato = INTERROTTO AND FuoriIngombroXNecessario) OR 
					Programma_J[J_PosFuoriIngombro].Stato = INTERROTTO THEN
						Ciclo^.Passo := 52;										
				ELSE
					IF StepInto THEN
						IF NOT FuoriIngombroXNecessario THEN
							Programma_X[X_PosStartLentaDepositoLastra].Stato 			:= DA_ESEGUIRE;
							Programma_X[X_PosStartLentaDepositoLastra].InterpolaAsse 	:= INTERPOLAZIONE_ASSE;
							ProgrammaToModule_X 										:= Programma_X[X_PosStartLentaDepositoLastra];
						END_IF
					
						Programma_Y[Y_PosStartLentaDepositoLastra].Stato 			:= DA_ESEGUIRE;
						Programma_Y[Y_PosStartLentaDepositoLastra].InterpolaAsse 	:= INTERPOLAZIONE_ASSE;
						ProgrammaToModule_Y 										:= Programma_Y[Y_PosStartLentaDepositoLastra];
						
						//Programma_Z[Z_PosStartLentaDepositoLastra].Stato 			:= DA_ESEGUIRE;
						//Programma_Z[Z_PosStartLentaDepositoLastra].InterpolaAsse 	:= INTERPOLAZIONE_ASSE;
						//ProgrammaToModule_Z 										:= Programma_Z[Z_PosStartLentaDepositoLastra];
					
					
						Programma_J[J_PosDepositoLastra].Stato 						:= DA_ESEGUIRE;
						Programma_J[J_PosDepositoLastra].InterpolaAsse 				:= INTERPOLAZIONE_ASSE;
						ProgrammaToModule_J 										:= Programma_J[J_PosDepositoLastra];
			
						StartInterpolazioneAssi^ := TRUE; //Abilito l'interpolazione degli assi

						Ciclo^.Passo := 53;
						STEPDone := FALSE;
					END_IF
				END_IF			
				
			(* Case 53 -  Attesa completamento del comando MOVETOPOS o del raggiungimento quota di Pre-Movimento se abilitata la funzione *)
			53: 
				IF Programma_X[X_PosStartLentaDepositoLastra].Stato = INTERROTTO OR
					Programma_Y[Y_PosStartLentaDepositoLastra].Stato = INTERROTTO OR
					Programma_Z[Z_PosFuoriIngombroCaricoLastra].Stato = INTERROTTO OR 
					Programma_J[J_PosDepositoLastra].Stato = INTERROTTO THEN
						Ciclo^.Passo := 53;
				ELSE	
					IF (Programma_Y[Y_PosStartLentaDepositoLastra].Stato = TERMINATO OR Asse_Y_InFinestraDiPassMode OR QuotaAnticipoDinamicaY_Raggiunta) AND
						(Programma_J[J_PosDepositoLastra].Stato = TERMINATO OR Asse_J_InFinestraDiPassMode OR QuotaAnticipoDinamicaJ_Raggiunta)  THEN 
							
							Ciclo^.Passo := 54;
							STEPDone := TRUE;							
					END_IF
				END_IF
				
			(* Case 54 - Vado a quota di START LENTA CON GLI ASSI Z*)
			54:
				IF Programma_X[X_PosStartLentaDepositoLastra].Stato = INTERROTTO OR
					Programma_Y[Y_PosStartLentaDepositoLastra].Stato = INTERROTTO OR
					//Programma_Z[Z_PosStartLentaDepositoLastra].Stato = INTERROTTO OR 
					Programma_J[J_PosDepositoLastra].Stato = INTERROTTO THEN
						Ciclo^.Passo := 54;										
				ELSE
					IF StepInto THEN
						Programma_Z[Z_PosStartLentaDepositoLastra].Stato 			:= DA_ESEGUIRE;
						Programma_Z[Z_PosStartLentaDepositoLastra].InterpolaAsse 	:= NO_INTERPOLAZIONE_ASSE;
						ProgrammaToModule_Z 										:= Programma_Z[Z_PosStartLentaDepositoLastra];
								
						Ciclo^.Passo := 55;
						STEPDone := FALSE;
					END_IF
				END_IF
			
			(* Case 55 - Attendo completamento comando o assi in finsetra *)
			55:
				IF Programma_Y[Y_PosStartLentaDepositoLastra].Stato = TERMINATO (*OR Asse_Y_InFinestraDiPassMode)*) AND 
					Programma_J[J_PosDepositoLastra].Stato = TERMINATO (*OR Asse_J_InFinestraDiPassMode)*) AND
					Programma_X[X_PosStartLentaDepositoLastra].Stato = TERMINATO (*OR Asse_X_InFinestraDiPassMode)*) AND 
					Programma_Z[Z_PosStartLentaDepositoLastra].Stato = TERMINATO OR Asse_Z_InFinestraDiPassMode THEN
						Ciclo^.Passo := 56;
						STEPDone := TRUE;
				ELSIF Programma_X[X_PosStartLentaDepositoLastra].Stato = INTERROTTO OR
					Programma_Y[Y_PosStartLentaDepositoLastra].Stato = INTERROTTO OR
					Programma_Z[Z_PosFuoriIngombroCaricoLastra].Stato = INTERROTTO OR 
					Programma_J[J_PosDepositoLastra].Stato = INTERROTTO THEN
						Ciclo^.Passo := 55;
				END_IF

			(* Case 56 - Vado a quota di finale con Y,Z,J *)
			56:
				IF Programma_X[X_PosStartLentaDepositoLastra].Stato = INTERROTTO OR
					Programma_Y[Y_PosFuoriIngombroCaricoLastra].Stato = INTERROTTO OR
					Programma_Z[Z_PosFuoriIngombroCaricoLastra].Stato = INTERROTTO OR 
					Programma_J[J_PosFuoriIngombro].Stato = INTERROTTO THEN
						Ciclo^.Passo := 56;										
				ELSE
					IF StepInto THEN
						TFParametersArrayClear(ADR(ParametersArray));
						Programma_Z[Z_PosDepositoInLentaLastra].Stato 			:= DA_ESEGUIRE;
						Programma_Z[Z_PosDepositoInLentaLastra].InterpolaAsse 	:= NO_INTERPOLAZIONE_ASSE;
						ProgrammaToModule_Z 									:= Programma_Z[Z_PosDepositoInLentaLastra];						
						Ciclo^.Passo := 57;
						STEPDone := FALSE;						
						//StartInterpolazioneAssi^ := TRUE; //Abilito l'interpolazione degli assi
						
					END_IF
				END_IF

			(* Case 57 - Attendo completamento comando o assi in finsetra *)
			57:
				IF //Programma_Y[Y_PosStartLentaDepositoLastra].Stato = TERMINATO (*OR Asse_Y_InFinestraDiPassMode)*) AND 
					//Programma_J[J_PosDepositoLastra].Stato = TERMINATO (*OR Asse_J_InFinestraDiPassMode)*) AND
					//Programma_X[X_PosStartLentaDepositoLastra].Stato = TERMINATO (*OR Asse_X_InFinestraDiPassMode)*) AND 
					Programma_Z[Z_PosDepositoInLentaLastra].Stato = TERMINATO (*OR Asse_Z_InFinestraDiPassMode)*) THEN
						Ciclo^.Passo := 90;
						STEPDone := TRUE;
				ELSIF //Programma_Y[Y_PosStartLentaDepositoLastra].Stato = INTERROTTO OR 
					//Programma_J[J_PosDepositoLastra].Stato = INTERROTTO OR 
					//Programma_X[X_PosStartLentaDepositoLastra].Stato = INTERROTTO OR
					Programma_Z[Z_PosDepositoInLentaLastra].Stato = INTERROTTO THEN
					Ciclo^.Passo := 57;								
				END_IF
						
		{endregion}	
			(* Case 90 - Attesa completamento posizionamento di tutti gli assi *)
			90: 
				IF TFStateCodeGet(ModulePinza^.State) = StateError THEN
					Ciclo^.Passo := 90;																
				ELSE
					IF StepInto THEN
						TFParametersArrayClear(ADR(ParametersArray));
						TFCommandSend(CmdUNLOAD,ParametersArray,ModulePinza^.Cmd);
						Ciclo^.Passo := 91;
						STEPDone := FALSE;
					END_IF							
				END_IF

			(* Case 91 - Attesa completamento rilascio pezzo *)	
			91:
				IF TFStateCodeGet(ModulePinza^.State) = StateError THEN
					Ciclo^.Passo := 91;																
				ELSE
					STEPDone := TRUE;
					IF TFStateCodeGet(ModulePinza^.State) = StateUNLOAD_END THEN//Pezzo rilasciato
						RichiestaDepositoALinea := FALSE;
						Ciclo^.Passo := 1000;//dichiaro il ciclo terminato
					END_IF	
				END_IF
			
			(* Case 1000 *)
			1000:
				RichiestaDepositoALinea := FALSE;
				StopDepositoPerArresto := FALSE;
				Ciclo^.Stato := TERMINATO;
				Ciclo^.Passo := 1000;
				
			(* Case 9999 - Ciclo NON annullato o NON terminato*)
			9999:
				Ciclo^.Stato := INTERROTTO;
				Ciclo^.Passo := 9999;
	ELSE						
		;
			
	END_CASE;
	(* controllo pinza in presa durante il ciclo *)  
	IF WorkAreaState[Mission.PPlace].Supporto.Tipologia <> CAVALLETTO AND WorkAreaState[Mission.PPlace].Supporto.Tipologia <> BUNDLE THEN
		IF Ciclo^.Passo >= 20 AND Ciclo^.Passo <= 90 THEN
			IF PinzaInPresa THEN
				 ;
			ELSE
				Errore := ErrLOADLOST;//Segnalo mancanza presenza pezzo
			END_IF
		END_IF
	ELSE
		IF Ciclo^.Passo >= 20 AND Ciclo^.Passo <= 42 THEN
			IF PinzaInPresa THEN
				 ;
			ELSE
				Errore := ErrLOADLOST;//Segnalo mancanza presenza pezzo
			END_IF
		END_IF
	END_IF
ELSE								//Se il ciclo deve essere interrotto, setto il suo nuovo stato
	Ciclo^.Stato := INTERROTTO;
END_IF

END_FUNCTION_BLOCK

// ---- POUs/TFCicliDiLavoro/Lastre/Cicli Depallettizzatore/TFCiclo_Prelievo_Lastra_Depal.TcPOU
FUNCTION_BLOCK TFCiclo_Prelievo_Lastra_Depal
VAR_INPUT
	Ciclo 		: POINTER TO Stato_Ciclo_Lavoro;
	Programma : POINTER TO TFProgramma_Ciclo_Lastra;
	ModuleAX_X : POINTER TO TFModulePalletizer_Ax;
	ModuleAX_Y : POINTER TO TFModulePalletizer_Ax;
	ModuleAX_Z : POINTER TO TFModulePalletizer_Ax;
	ModuleAX_J : POINTER TO TFModulePalletizer_AxJ_Lastre;
	ModulePinza : POINTER TO TFModulePalletizer_Pinza;
	StartInterpolazioneAssi : POINTER TO BOOL;
	QuotaPassModePuntoIntermedio : ARRAY [1..3] OF REAL;
	AbilitazioneGlobalePassMode	: BOOL;
	InterrompiCiclo : BOOL;
	Abilita_Ciclo_Step : BOOL;
	Command_Step : BOOL;
	AbilitazioneAnticipoDinamicoMovimenti : BOOL;
	PrelievoPezzoOrizzontale : BOOL;//indica che il prelievo del pezzo è orizzontale, sono su pallet o cassa
	NumeroTentativiPresa : UINT := 2;//Numero dei tentativi da effettuare prima di eliminare l'elemento
END_VAR
VAR_OUTPUT
	STEPDone	: BOOL;
	SupportoVuoto : BOOL;
	Errore : UINT;
END_VAR
VAR
	StepInto : BOOL;
	NumeroTentativiPresaAttuali : UINT;
	TimerAttesaCadutaLastra : REAL;
	i: UINT;
	RichiestaEspulsionePerPolistirolo: BOOL;
	PipickOld : uint;
END_VAR


TFTimerCall(ADR(TimerAttesaCadutaLastra),TimeBase);
(* Set della variabile che mi permette di fare lo STEP nel ciclo *)
StepInto := (Abilita_Ciclo_Step AND Command_Step) OR NOT Abilita_Ciclo_Step;

(* Reset Anticipo Dinamico se non ho l'abilitazione *)
IF NOT AbilitazioneAnticipoDinamicoMovimenti  OR NOT HMI_DisabilitaAnticipiGLOBALE THEN
	QuotaAnticipoDinamicaX_Raggiunta := FALSE;
	QuotaAnticipoDinamicaY_Raggiunta := FALSE;
	QuotaAnticipoDinamicaZ_Raggiunta := FALSE;
END_IF

IF NOT InterrompiCiclo THEN
	IF Ciclo^.Stato = TERMINATO OR Ciclo^.Stato = ANNULLATO THEN
		Ciclo^.Passo := 0;
		Errore := 0;
	ELSIF Ciclo^.Stato = INTERROTTO THEN
		Ciclo^.Passo := 999;
	END_IF
	Errore := 0;
	Ciclo^.Stato := IN_ESECUZIONE;
	CASE Ciclo^.Passo OF
			(* Case 0 *)
			0:  Ciclo^.Stato := IN_ESECUZIONE;
				Ciclo^.Passo := 10;
				STEPDone := FALSE;
				SupportoVuoto := FALSE;
				NumeroTentativiPresaAttuali := 0;
				IF Mission.PPick <> PipickOld THEN
					idxTasteg := 0;
					MemoriaQuoteTasteggio := MemoriaQuoteTasteggioVuoto;
					RichiestaEspulsionePerPolistirolo := FALSE;
				END_IF
				PipickOld := Mission.PPick;
				
			(* Case 10 - Spengo aspirazione *)
			10:	IF ModulePinza^.CmdNext.Code = '' THEN
					TFParametersArrayClear(ADR(ParametersArray));
					TFCommandSend(CmdUNLOAD,ParametersArray,ModulePinza^.Cmd);
					Ciclo^.Passo := 11;
				END_IF

			(* Case 11 - Attesa Aspirazione spenta *)
			11:
				IF TFStateCodeGet(ModulePinza^.State) = StateUNLOAD_END THEN
					Ciclo^.Passo := 20;
				END_IF
						
